LIN {X 0,Y 572.938,Z 557.197,A -85,B 0,C 180,E1 -2247.891,E2 -2247.891} C_VEL
LIN {X 0,Y 572.94,Z 558.785,A -85,B 0,C 180,E1 -2249.297,E2 -2249.297} C_VEL
LIN {X 0,Y 572.938,Z 559,A -85,B 0,C 180,E1 -2250,E2 -2250} C_VEL
LIN {X 0,Y 572.946,Z 558.187,A -85,B 0,C 180,E1 -2251.406,E2 -2251.406} C_VEL
LIN {X 0,Y 572.938,Z 557.2,A -85,B 0,C 180,E1 -2252.109,E2 -2252.109} C_VEL
LIN {X 0,Y 572.959,Z 555.811,A -85,B 0,C 180,E1 -2252.812,E2 -2252.812} C_VEL
LIN {X 0,Y 573.014,Z 552.897,A -85,B 0,C 180,E1 -2253.868,E2 -2253.868} C_VEL
LIN {X 0,Y 572.963,Z 548.95,A -85,B 0,C 180,E1 -2254.925,E2 -2254.925} C_VEL
LIN {X 0,Y 573.068,Z 542.878,A -85,B 0,C 180,E1 -2256.16,E2 -2256.16} C_VEL
LIN {X 0,Y 573.119,Z 536.24,A -85,B 0,C 180,E1 -2257.22,E2 -2257.22} C_VEL
LIN {X 0,Y 573.192,Z 527.993,A -85,B 0,C 180,E1 -2258.283,E2 -2258.283} C_VEL
LIN {X 0,Y 573.319,Z 517.605,A -85,B 0,C 180,E1 -2259.347,E2 -2259.347} C_VEL
LIN {X 0,Y 573.431,Z 507.929,A -85,B 0,C 180,E1 -2260.147,E2 -2260.147} C_VEL
LIN {X 0,Y 573.549,Z 497.407,A -85,B 0,C 180,E1 -2260.854,E2 -2260.854} C_VEL
LIN {X 0,Y 573.652,Z 486.294,A -85,B 0,C 180,E1 -2261.447,E2 -2261.447} C_VEL
LIN {X 0,Y 573.694,Z 474.482,A -85,B 0,C 180,E1 -2261.93,E2 -2261.93} C_VEL
LIN {X 0,Y 573.799,Z 461.448,A -85,B 0,C 180,E1 -2262.309,E2 -2262.309} C_VEL
LIN {X 0,Y 573.915,Z 449.111,A -85,B 0,C 180,E1 -2262.531,E2 -2262.531} C_VEL
LIN {X 0,Y 573.909,Z 350.304,A -85,B 0,C 180,E1 -2263.775,E2 -2263.775} C_VEL
LIN {X 0,Y 573.398,Z 346.616,A -85,B 0,C 180,E1 -2263.85,E2 -2263.85} C_VEL
LIN {X 0,Y 573.568,Z 326.122,A -85,B 0,C 180,E1 -2266.727,E2 -2266.727} C_VEL
LIN {X 0,Y 573.803,Z 305.614,A -85,B 0,C 180,E1 -2269.646,E2 -2269.646} C_VEL
LIN {X 0,Y 574.043,Z 285.773,A -85,B 0,C 180,E1 -2272.494,E2 -2272.494} C_VEL
LIN {X 0,Y 573.587,Z 280.817,A -85,B 0,C 180,E1 -2273.226,E2 -2273.226} C_VEL
LIN {X 0,Y 573.252,Z 279.081,A -85,B 0,C 180,E1 -2273.496,E2 -2273.496} C_VEL
LIN {X 0,Y 573.261,Z 279.078,A -85,B 0,C 180,E1 -2276.189,E2 -2276.189} C_VEL
LIN {X 0,Y 573.237,Z 279.077,A -85,B 0,C 180,E1 -2278.564,E2 -2278.564} C_VEL
LIN {X 0,Y 573.226,Z 279.075,A -85,B 0,C 180,E1 -2280.993,E2 -2280.993} C_VEL
LIN {X 0,Y 573.262,Z 279.072,A -85,B 0,C 180,E1 -2283.523,E2 -2283.523} C_VEL
LIN {X 0,Y 573.213,Z 279.084,A -85,B 0,C 180,E1 -2286.051,E2 -2286.051} C_VEL
LIN {X 0,Y 573.24,Z 279.077,A -85,B 0,C 180,E1 -2288.701,E2 -2288.701} C_VEL
LIN {X 0,Y 573.252,Z 279.072,A -85,B 0,C 180,E1 -2291.595,E2 -2291.595} C_VEL
LIN {X 0,Y 573.226,Z 279.083,A -85,B 0,C 180,E1 -2294.334,E2 -2294.334} C_VEL
LIN {X 0,Y 573.238,Z 279.074,A -85,B 0,C 180,E1 -2297.358,E2 -2297.358} C_VEL
LIN {X 0,Y 573.237,Z 279.08,A -85,B 0,C 180,E1 -2300.392,E2 -2300.392} C_VEL
LIN {X 0,Y 573.25,Z 279.076,A -85,B 0,C 180,E1 -2303.077,E2 -2303.077} C_VEL
LIN {X 0,Y 573.263,Z 279.07,A -85,B 0,C 180,E1 -2305.671,E2 -2305.671} C_VEL
LIN {X 0,Y 573.245,Z 279.074,A -85,B 0,C 180,E1 -2308.185,E2 -2308.185} C_VEL
LIN {X 0,Y 573.261,Z 279.076,A -85,B 0,C 180,E1 -2310.634,E2 -2310.634} C_VEL
LIN {X 0,Y 573.248,Z 279.083,A -85,B 0,C 180,E1 -2313.024,E2 -2313.024} C_VEL
LIN {X 0,Y 573.271,Z 279.075,A -85,B 0,C 180,E1 -2315.366,E2 -2315.366} C_VEL
LIN {X 0,Y 573.223,Z 279.076,A -85,B 0,C 180,E1 -2318.419,E2 -2318.419} C_VEL
LIN {X 0,Y 573.274,Z 279.072,A -85,B 0,C 180,E1 -2320.728,E2 -2320.728} C_VEL
LIN {X 0,Y 573.244,Z 279.077,A -85,B 0,C 180,E1 -2323.621,E2 -2323.621} C_VEL
LIN {X 0,Y 573.267,Z 279.073,A -85,B 0,C 180,E1 -2325.807,E2 -2325.807} C_VEL
LIN {X 0,Y 573.257,Z 279.072,A -85,B 0,C 180,E1 -2328.745,E2 -2328.745} C_VEL
LIN {X 0,Y 573.284,Z 279.078,A -85,B 0,C 180,E1 -2331.54,E2 -2331.54} C_VEL
LIN {X 0,Y 573.284,Z 279.068,A -85,B 0,C 180,E1 -2334.372,E2 -2334.372} C_VEL
LIN {X 0,Y 573.297,Z 279.073,A -85,B 0,C 180,E1 -2337.892,E2 -2337.892} C_VEL
LIN {X 0,Y 573.321,Z 279.063,A -85,B 0,C 180,E1 -2340.702,E2 -2340.702} C_VEL
LIN {X 0,Y 573.238,Z 279.079,A -85,B 0,C 180,E1 -2343.514,E2 -2343.514} C_VEL
LIN {X 0,Y 573.29,Z 279.073,A -85,B 0,C 180,E1 -2345.628,E2 -2345.628} C_VEL
LIN {X 0,Y 573.277,Z 279.071,A -85,B 0,C 180,E1 -2348.459,E2 -2348.459} C_VEL
LIN {X 0,Y 573.266,Z 279.071,A -85,B 0,C 180,E1 -2351.312,E2 -2351.312} C_VEL
LIN {X 0,Y 573.253,Z 279.081,A -85,B 0,C 180,E1 -2354.193,E2 -2354.193} C_VEL
LIN {X 0,Y 573.252,Z 279.072,A -85,B 0,C 180,E1 -2357.112,E2 -2357.112} C_VEL
LIN {X 0,Y 573.235,Z 279.081,A -85,B 0,C 180,E1 -2360.077,E2 -2360.077} C_VEL
LIN {X 0,Y 573.227,Z 279.086,A -85,B 0,C 180,E1 -2362.338,E2 -2362.338} C_VEL
LIN {X 0,Y 573.24,Z 279.077,A -85,B 0,C 180,E1 -2364.37,E2 -2364.37} C_VEL
LIN {X 0,Y 572.61,Z 279.158,A -85,B 0,C 180,E1 -2364.956,E2 -2364.956} C_VEL
LIN {X 0,Y 569.752,Z 279.513,A -85,B 0,C 180,E1 -2365.907,E2 -2365.907} C_VEL
LIN {X 0,Y 567.309,Z 279.819,A -85,B 0,C 180,E1 -2366.672,E2 -2366.672} C_VEL
LIN {X 0,Y 566.252,Z 279.944,A -85,B 0,C 180,E1 -2367.264,E2 -2367.264} C_VEL
LIN {X 0,Y 566.163,Z 279.955,A -85,B 0,C 180,E1 -2367.464,E2 -2367.464} C_VEL
LIN {X 0,Y 566.194,Z 279.951,A -85,B 0,C 180,E1 -2369.769,E2 -2369.769} C_VEL
LIN {X 0,Y 566.198,Z 279.958,A -85,B 0,C 180,E1 -2372.43,E2 -2372.43} C_VEL
LIN {X 0,Y 566.173,Z 279.959,A -85,B 0,C 180,E1 -2374.99,E2 -2374.99} C_VEL
LIN {X 0,Y 566.19,Z 279.952,A -85,B 0,C 180,E1 -2377.461,E2 -2377.461} C_VEL
LIN {X 0,Y 566.201,Z 279.952,A -85,B 0,C 180,E1 -2380.2,E2 -2380.2} C_VEL
LIN {X 0,Y 566.192,Z 279.959,A -85,B 0,C 180,E1 -2383.055,E2 -2383.055} C_VEL
LIN {X 0,Y 566.188,Z 279.951,A -85,B 0,C 180,E1 -2386.05,E2 -2386.05} C_VEL
LIN {X 0,Y 566.198,Z 279.959,A -85,B 0,C 180,E1 -2389.215,E2 -2389.215} C_VEL
LIN {X 0,Y 566.175,Z 279.956,A -85,B 0,C 180,E1 -2391.637,E2 -2391.637} C_VEL
LIN {X 0,Y 566.157,Z 279.955,A -85,B 0,C 180,E1 -2394.308,E2 -2394.308} C_VEL
LIN {X 0,Y 566.194,Z 279.955,A -85,B 0,C 180,E1 -2396.897,E2 -2396.897} C_VEL
LIN {X 0,Y 566.159,Z 279.965,A -85,B 0,C 180,E1 -2399.407,E2 -2399.407} C_VEL
LIN {X 0,Y 566.184,Z 279.955,A -85,B 0,C 180,E1 -2401.856,E2 -2401.856} C_VEL
LIN {X 0,Y 566.18,Z 279.953,A -85,B 0,C 180,E1 -2404.25,E2 -2404.25} C_VEL
LIN {X 0,Y 566.172,Z 279.961,A -85,B 0,C 180,E1 -2407.369,E2 -2407.369} C_VEL
LIN {X 0,Y 566.202,Z 279.96,A -85,B 0,C 180,E1 -2409.663,E2 -2409.663} C_VEL
LIN {X 0,Y 566.175,Z 279.96,A -85,B 0,C 180,E1 -2411.921,E2 -2411.921} C_VEL
LIN {X 0,Y 566.188,Z 279.952,A -85,B 0,C 180,E1 -2414.891,E2 -2414.891} C_VEL
LIN {X 0,Y 566.209,Z 279.96,A -85,B 0,C 180,E1 -2417.819,E2 -2417.819} C_VEL
LIN {X 0,Y 566.179,Z 279.957,A -85,B 0,C 180,E1 -2420.714,E2 -2420.714} C_VEL
LIN {X 0,Y 566.192,Z 280.141,A -85,B 0,C 180,E1 -2420.894,E2 -2420.894} C_VEL
LIN {X 0,Y 566.476,Z 285.072,A -85,B 0,C 180,E1 -2421.798,E2 -2421.798} C_VEL
LIN {X 0,Y 566.29,Z 300.723,A -85,B 0,C 180,E1 -2424.66,E2 -2424.66} C_VEL
LIN {X 0,Y 566.196,Z 308.354,A -85,B 0,C 180,E1 -2426.041,E2 -2426.041} C_VEL
LIN {X 0,Y 567.175,Z 314.722,A -85,B 0,C 180,E1 -2426.159,E2 -2426.159} C_VEL
LIN {X 0,Y 566.923,Z 414.925,A -85,B 0,C 180,E1 -2427.447,E2 -2427.447} C_VEL
LIN {X 0,Y 566.838,Z 428.007,A -85,B 0,C 180,E1 -2427.758,E2 -2427.758} C_VEL
LIN {X 0,Y 566.75,Z 441.122,A -85,B 0,C 180,E1 -2428.224,E2 -2428.224} C_VEL
LIN {X 0,Y 566.61,Z 452.221,A -85,B 0,C 180,E1 -2428.756,E2 -2428.756} C_VEL
LIN {X 0,Y 566.39,Z 463.741,A -85,B 0,C 180,E1 -2429.467,E2 -2429.467} C_VEL
LIN {X 0,Y 566.297,Z 474.096,A -85,B 0,C 180,E1 -2430.267,E2 -2430.267} C_VEL
LIN {X 0,Y 566.199,Z 482.596,A -85,B 0,C 180,E1 -2431.067,E2 -2431.067} C_VEL
LIN {X 0,Y 566.087,Z 490.471,A -85,B 0,C 180,E1 -2431.957,E2 -2431.957} C_VEL
LIN {X 0,Y 566.044,Z 498.203,A -85,B 0,C 180,E1 -2433.025,E2 -2433.025} C_VEL
LIN {X 0,Y 565.964,Z 505.322,A -85,B 0,C 180,E1 -2434.273,E2 -2434.273} C_VEL
LIN {X 0,Y 565.923,Z 510.091,A -85,B 0,C 180,E1 -2435.344,E2 -2435.344} C_VEL
LIN {X 0,Y 565.944,Z 514.182,A -85,B 0,C 180,E1 -2436.56,E2 -2436.56} C_VEL
LIN {X 0,Y 565.876,Z 517.108,A -85,B 0,C 180,E1 -2437.852,E2 -2437.852} C_VEL
LIN {X 0,Y 565.851,Z 518.129,A -85,B 0,C 180,E1 -2438.572,E2 -2438.572} C_VEL
LIN {X 0,Y 565.88,Z 518.998,A -85,B 0,C 180,E1 -2440.013,E2 -2440.013} C_VEL
LIN {X 0,Y 565.9,Z 518.518,A -85,B 0,C 180,E1 -2441.154,E2 -2441.154} C_VEL
LIN {X 0,Y 565.867,Z 517.182,A -85,B 0,C 180,E1 -2442.189,E2 -2442.189} C_VEL
LIN {X 0,Y 565.852,Z 515.747,A -85,B 0,C 180,E1 -2442.919,E2 -2442.919} C_VEL
LIN {X 0,Y 565.916,Z 512.727,A -85,B 0,C 180,E1 -2444.015,E2 -2444.015} C_VEL
LIN {X 0,Y 565.947,Z 508.595,A -85,B 0,C 180,E1 -2445.117,E2 -2445.117} C_VEL
LIN {X 0,Y 565.955,Z 502.16,A -85,B 0,C 180,E1 -2446.41,E2 -2446.41} C_VEL
LIN {X 0,Y 566.076,Z 495.095,A -85,B 0,C 180,E1 -2447.522,E2 -2447.522} C_VEL
LIN {X 0,Y 566.142,Z 487.805,A -85,B 0,C 180,E1 -2448.455,E2 -2448.455} C_VEL
LIN {X 0,Y 566.249,Z 477.889,A -85,B 0,C 180,E1 -2449.484,E2 -2449.484} C_VEL
LIN {X 0,Y 566.378,Z 467.78,A -85,B 0,C 180,E1 -2450.331,E2 -2450.331} C_VEL
LIN {X 0,Y 566.526,Z 456.576,A -85,B 0,C 180,E1 -2451.085,E2 -2451.085} C_VEL
LIN {X 0,Y 566.679,Z 444.223,A -85,B 0,C 180,E1 -2451.73,E2 -2451.73} C_VEL
LIN {X 0,Y 566.776,Z 431.645,A -85,B 0,C 180,E1 -2452.222,E2 -2452.222} C_VEL
LIN {X 0,Y 566.799,Z 419.367,A -85,B 0,C 180,E1 -2452.557,E2 -2452.557} C_VEL
LIN {X 0,Y 566.916,Z 402.556,A -85,B 0,C 180,E1 -2452.817,E2 -2452.817} C_VEL
LIN {X 0,Y 567.066,Z 313.669,A -85,B 0,C 180,E1 -2453.947,E2 -2453.947} C_VEL
LIN {X 0,Y 566.196,Z 308.415,A -85,B 0,C 180,E1 -2454.038,E2 -2454.038} C_VEL
LIN {X 0,Y 566.375,Z 293.793,A -85,B 0,C 180,E1 -2456.693,E2 -2456.693} C_VEL
LIN {X 0,Y 566.454,Z 281.463,A -85,B 0,C 180,E1 -2458.939,E2 -2458.939} C_VEL
LIN {X 0,Y 566.256,Z 279.95,A -85,B 0,C 180,E1 -2459.255,E2 -2459.255} C_VEL
LIN {X 0,Y 566.204,Z 279.959,A -85,B 0,C 180,E1 -2462.43,E2 -2462.43} C_VEL
LIN {X 0,Y 566.178,Z 279.955,A -85,B 0,C 180,E1 -2464.989,E2 -2464.989} C_VEL
LIN {X 0,Y 566.195,Z 279.95,A -85,B 0,C 180,E1 -2467.461,E2 -2467.461} C_VEL
LIN {X 0,Y 566.206,Z 279.956,A -85,B 0,C 180,E1 -2470.199,E2 -2470.199} C_VEL
LIN {X 0,Y 566.199,Z 279.954,A -85,B 0,C 180,E1 -2473.054,E2 -2473.054} C_VEL
LIN {X 0,Y 566.193,Z 279.953,A -85,B 0,C 180,E1 -2476.049,E2 -2476.049} C_VEL
LIN {X 0,Y 566.203,Z 279.953,A -85,B 0,C 180,E1 -2479.215,E2 -2479.215} C_VEL
LIN {X 0,Y 566.185,Z 279.952,A -85,B 0,C 180,E1 -2481.637,E2 -2481.637} C_VEL
LIN {X 0,Y 566.161,Z 279.956,A -85,B 0,C 180,E1 -2484.308,E2 -2484.308} C_VEL
LIN {X 0,Y 566.218,Z 279.956,A -85,B 0,C 180,E1 -2486.898,E2 -2486.898} C_VEL
LIN {X 0,Y 566.18,Z 279.957,A -85,B 0,C 180,E1 -2489.407,E2 -2489.407} C_VEL
LIN {X 0,Y 566.21,Z 279.948,A -85,B 0,C 180,E1 -2491.857,E2 -2491.857} C_VEL
LIN {X 0,Y 566.212,Z 279.948,A -85,B 0,C 180,E1 -2494.251,E2 -2494.251} C_VEL
LIN {X 0,Y 566.172,Z 279.954,A -85,B 0,C 180,E1 -2496.718,E2 -2496.718} C_VEL
LIN {X 0,Y 566.207,Z 279.954,A -85,B 0,C 180,E1 -2499.663,E2 -2499.663} C_VEL
LIN {X 0,Y 566.198,Z 279.951,A -85,B 0,C 180,E1 -2502.668,E2 -2502.668} C_VEL
LIN {X 0,Y 566.233,Z 279.957,A -85,B 0,C 180,E1 -2505.627,E2 -2505.627} C_VEL
LIN {X 0,Y 566.233,Z 279.945,A -85,B 0,C 180,E1 -2508.675,E2 -2508.675} C_VEL
LIN {X 0,Y 566.226,Z 279.952,A -85,B 0,C 180,E1 -2511.434,E2 -2511.434} C_VEL
LIN {X 0,Y 566.256,Z 279.946,A -85,B 0,C 180,E1 -2514.302,E2 -2514.302} C_VEL
LIN {X 0,Y 566.281,Z 279.949,A -85,B 0,C 180,E1 -2517.866,E2 -2517.866} C_VEL
LIN {X 0,Y 566.299,Z 279.939,A -85,B 0,C 180,E1 -2520.711,E2 -2520.711} C_VEL
LIN {X 0,Y 566.27,Z 279.941,A -85,B 0,C 180,E1 -2522.846,E2 -2522.846} C_VEL
LIN {X 0,Y 566.256,Z 279.946,A -85,B 0,C 180,E1 -2525.698,E2 -2525.698} C_VEL
LIN {X 0,Y 566.226,Z 279.953,A -85,B 0,C 180,E1 -2528.566,E2 -2528.566} C_VEL
LIN {X 0,Y 566.242,Z 279.944,A -85,B 0,C 180,E1 -2531.454,E2 -2531.454} C_VEL
LIN {X 0,Y 566.234,Z 279.956,A -85,B 0,C 180,E1 -2534.507,E2 -2534.507} C_VEL
LIN {X 0,Y 566.199,Z 279.951,A -85,B 0,C 180,E1 -2537.332,E2 -2537.332} C_VEL
LIN {X 0,Y 566.207,Z 279.954,A -85,B 0,C 180,E1 -2540.338,E2 -2540.338} C_VEL
LIN {X 0,Y 566.173,Z 279.956,A -85,B 0,C 180,E1 -2543.282,E2 -2543.282} C_VEL
LIN {X 0,Y 566.214,Z 279.948,A -85,B 0,C 180,E1 -2545.749,E2 -2545.749} C_VEL
LIN {X 0,Y 566.203,Z 279.95,A -85,B 0,C 180,E1 -2548.202,E2 -2548.202} C_VEL
LIN {X 0,Y 566.191,Z 279.96,A -85,B 0,C 180,E1 -2551.077,E2 -2551.077} C_VEL
LIN {X 0,Y 566.212,Z 279.95,A -85,B 0,C 180,E1 -2553.734,E2 -2553.734} C_VEL
LIN {X 0,Y 566.2,Z 279.951,A -85,B 0,C 180,E1 -2556.57,E2 -2556.57} C_VEL
LIN {X 0,Y 566.216,Z 279.949,A -85,B 0,C 180,E1 -2559.686,E2 -2559.686} C_VEL
LIN {X 0,Y 566.203,Z 279.953,A -85,B 0,C 180,E1 -2562.917,E2 -2562.917} C_VEL
LIN {X 0,Y 566.195,Z 279.953,A -85,B 0,C 180,E1 -2566.049,E2 -2566.049} C_VEL
LIN {X 0,Y 566.205,Z 279.955,A -85,B 0,C 180,E1 -2569.215,E2 -2569.215} C_VEL
LIN {X 0,Y 566.187,Z 279.962,A -85,B 0,C 180,E1 -2571.637,E2 -2571.637} C_VEL
LIN {X 0,Y 566.163,Z 279.957,A -85,B 0,C 180,E1 -2574.308,E2 -2574.308} C_VEL
LIN {X 0,Y 566.207,Z 279.95,A -85,B 0,C 180,E1 -2576.897,E2 -2576.897} C_VEL
LIN {X 0,Y 566.183,Z 279.957,A -85,B 0,C 180,E1 -2579.407,E2 -2579.407} C_VEL
LIN {X 0,Y 566.197,Z 279.961,A -85,B 0,C 180,E1 -2581.857,E2 -2581.857} C_VEL
LIN {X 0,Y 566.211,Z 279.957,A -85,B 0,C 180,E1 -2584.251,E2 -2584.251} C_VEL
LIN {X 0,Y 566.227,Z 280.119,A -85,B 0,C 180,E1 -2586.404,E2 -2586.404} C_VEL
LIN {X 0,Y 567.053,Z 285.451,A -85,B 0,C 180,E1 -2587.213,E2 -2587.213} C_VEL
LIN {X 0,Y 566.869,Z 303.945,A -85,B 0,C 180,E1 -2589.877,E2 -2589.877} C_VEL
LIN {X 0,Y 566.611,Z 324.891,A -85,B 0,C 180,E1 -2592.885,E2 -2592.885} C_VEL
LIN {X 0,Y 566.39,Z 346.612,A -85,B 0,C 180,E1 -2595.974,E2 -2595.974} C_VEL
LIN {X 0,Y 567.217,Z 352.273,A -85,B 0,C 180,E1 -2596.084,E2 -2596.084} C_VEL
LIN {X 0,Y 566.954,Z 454.939,A -85,B 0,C 180,E1 -2597.403,E2 -2597.403} C_VEL
LIN {X 0,Y 566.847,Z 467.451,A -85,B 0,C 180,E1 -2597.696,E2 -2597.696} C_VEL
LIN {X 0,Y 566.724,Z 480.373,A -85,B 0,C 180,E1 -2598.148,E2 -2598.148} C_VEL
LIN {X 0,Y 566.631,Z 492.046,A -85,B 0,C 180,E1 -2598.702,E2 -2598.702} C_VEL
LIN {X 0,Y 566.488,Z 502.905,A -85,B 0,C 180,E1 -2599.365,E2 -2599.365} C_VEL
LIN {X 0,Y 566.33,Z 513.537,A -85,B 0,C 180,E1 -2600.175,E2 -2600.175} C_VEL
LIN {X 0,Y 566.206,Z 523.081,A -85,B 0,C 180,E1 -2601.074,E2 -2601.074} C_VEL
LIN {X 0,Y 566.111,Z 530.959,A -85,B 0,C 180,E1 -2601.971,E2 -2601.971} C_VEL
LIN {X 0,Y 566.004,Z 538.621,A -85,B 0,C 180,E1 -2603.046,E2 -2603.046} C_VEL
LIN {X 0,Y 566.004,Z 545.679,A -85,B 0,C 180,E1 -2604.299,E2 -2604.299} C_VEL
LIN {X 0,Y 565.933,Z 550.371,A -85,B 0,C 180,E1 -2605.37,E2 -2605.37} C_VEL
LIN {X 0,Y 565.927,Z 553.957,A -85,B 0,C 180,E1 -2606.44,E2 -2606.44} C_VEL
LIN {X 0,Y 565.878,Z 555.807,A -85,B 0,C 180,E1 -2607.152,E2 -2607.152} C_VEL
LIN {X 0,Y 565.845,Z 558.185,A -85,B 0,C 180,E1 -2608.576,E2 -2608.576} C_VEL
LIN {X 0,Y 565.839,Z 559,A -85,B 0,C 180,E1 -2610,E2 -2610} C_VEL
LIN {X 0,Y 565.845,Z 558.186,A -85,B 0,C 180,E1 -2611.423,E2 -2611.423} C_VEL
LIN {X 0,Y 565.878,Z 555.811,A -85,B 0,C 180,E1 -2612.847,E2 -2612.847} C_VEL
LIN {X 0,Y 565.926,Z 552.896,A -85,B 0,C 180,E1 -2613.916,E2 -2613.916} C_VEL
LIN {X 0,Y 565.878,Z 548.95,A -85,B 0,C 180,E1 -2614.987,E2 -2614.987} C_VEL
LIN {X 0,Y 566.004,Z 543.869,A -85,B 0,C 180,E1 -2616.058,E2 -2616.058} C_VEL
LIN {X 0,Y 566.04,Z 537.47,A -85,B 0,C 180,E1 -2617.132,E2 -2617.132} C_VEL
LIN {X 0,Y 566.128,Z 529.481,A -85,B 0,C 180,E1 -2618.207,E2 -2618.207} C_VEL
LIN {X 0,Y 566.228,Z 521.338,A -85,B 0,C 180,E1 -2619.105,E2 -2619.105} C_VEL
LIN {X 0,Y 566.336,Z 511.404,A -85,B 0,C 180,E1 -2620.005,E2 -2620.005} C_VEL
LIN {X 0,Y 566.543,Z 500.307,A -85,B 0,C 180,E1 -2620.806,E2 -2620.806} C_VEL
LIN {X 0,Y 566.64,Z 489.182,A -85,B 0,C 180,E1 -2621.446,E2 -2621.446} C_VEL
LIN {X 0,Y 566.757,Z 476.99,A -85,B 0,C 180,E1 -2621.987,E2 -2621.987} C_VEL
LIN {X 0,Y 566.868,Z 464.19,A -85,B 0,C 180,E1 -2622.394,E2 -2622.394} C_VEL
LIN {X 0,Y 566.986,Z 450.626,A -85,B 0,C 180,E1 -2622.664,E2 -2622.664} C_VEL
LIN {X 0,Y 567.103,Z 351.644,A -85,B 0,C 180,E1 -2623.927,E2 -2623.927} C_VEL
LIN {X 0,Y 566.406,Z 346.616,A -85,B 0,C 180,E1 -2624.025,E2 -2624.025} C_VEL
LIN {X 0,Y 566.606,Z 324.043,A -85,B 0,C 180,E1 -2627.237,E2 -2627.237} C_VEL
LIN {X 0,Y 566.868,Z 303.962,A -85,B 0,C 180,E1 -2630.123,E2 -2630.123} C_VEL
LIN {X 0,Y 567.088,Z 285.517,A -85,B 0,C 180,E1 -2632.785,E2 -2632.785} C_VEL
LIN {X 0,Y 566.214,Z 279.959,A -85,B 0,C 180,E1 -2633.645,E2 -2633.645} C_VEL
LIN {X 0,Y 566.21,Z 279.958,A -85,B 0,C 180,E1 -2635.749,E2 -2635.749} C_VEL
LIN {X 0,Y 566.203,Z 279.959,A -85,B 0,C 180,E1 -2638.201,E2 -2638.201} C_VEL
LIN {X 0,Y 566.191,Z 279.951,A -85,B 0,C 180,E1 -2641.076,E2 -2641.076} C_VEL
LIN {X 0,Y 566.211,Z 279.952,A -85,B 0,C 180,E1 -2643.734,E2 -2643.734} C_VEL
LIN {X 0,Y 566.199,Z 279.956,A -85,B 0,C 180,E1 -2646.569,E2 -2646.569} C_VEL
LIN {X 0,Y 566.213,Z 279.95,A -85,B 0,C 180,E1 -2649.685,E2 -2649.685} C_VEL
LIN {X 0,Y 566.212,Z 279.954,A -85,B 0,C 180,E1 -2652.087,E2 -2652.087} C_VEL
LIN {X 0,Y 566.169,Z 279.956,A -85,B 0,C 180,E1 -2655.035,E2 -2655.035} C_VEL
LIN {X 0,Y 566.216,Z 279.951,A -85,B 0,C 180,E1 -2658.135,E2 -2658.135} C_VEL
LIN {X 0,Y 566.212,Z 279.958,A -85,B 0,C 180,E1 -2660.726,E2 -2660.726} C_VEL
LIN {X 0,Y 566.182,Z 279.952,A -85,B 0,C 180,E1 -2663.787,E2 -2663.787} C_VEL
LIN {X 0,Y 566.208,Z 279.951,A -85,B 0,C 180,E1 -2666.265,E2 -2666.265} C_VEL
LIN {X 0,Y 566.196,Z 279.961,A -85,B 0,C 180,E1 -2668.922,E2 -2668.922} C_VEL
LIN {X 0,Y 566.207,Z 279.949,A -85,B 0,C 180,E1 -2671.857,E2 -2671.857} C_VEL
LIN {X 0,Y 566.211,Z 279.949,A -85,B 0,C 180,E1 -2674.251,E2 -2674.251} C_VEL
LIN {X 0,Y 566.187,Z 279.956,A -85,B 0,C 180,E1 -2676.713,E2 -2676.713} C_VEL
LIN {X 0,Y 566.208,Z 279.952,A -85,B 0,C 180,E1 -2679.662,E2 -2679.662} C_VEL
LIN {X 0,Y 566.194,Z 279.953,A -85,B 0,C 180,E1 -2682.668,E2 -2682.668} C_VEL
LIN {X 0,Y 566.228,Z 279.952,A -85,B 0,C 180,E1 -2685.626,E2 -2685.626} C_VEL
LIN {X 0,Y 566.229,Z 279.947,A -85,B 0,C 180,E1 -2688.675,E2 -2688.675} C_VEL
LIN {X 0,Y 566.228,Z 279.957,A -85,B 0,C 180,E1 -2691.434,E2 -2691.434} C_VEL
LIN {X 0,Y 566.251,Z 279.944,A -85,B 0,C 180,E1 -2694.301,E2 -2694.301} C_VEL
LIN {X 0,Y 566.269,Z 279.949,A -85,B 0,C 180,E1 -2697.866,E2 -2697.866} C_VEL
LIN {X 0,Y 566.292,Z 279.939,A -85,B 0,C 180,E1 -2700.711,E2 -2700.711} C_VEL
LIN {X 0,Y 566.263,Z 279.942,A -85,B 0,C 180,E1 -2702.845,E2 -2702.845} C_VEL
LIN {X 0,Y 566.256,Z 279.951,A -85,B 0,C 180,E1 -2705.698,E2 -2705.698} C_VEL
LIN {X 0,Y 566.221,Z 279.949,A -85,B 0,C 180,E1 -2708.566,E2 -2708.566} C_VEL
LIN {X 0,Y 566.236,Z 279.947,A -85,B 0,C 180,E1 -2711.454,E2 -2711.454} C_VEL
LIN {X 0,Y 566.217,Z 279.952,A -85,B 0,C 180,E1 -2714.502,E2 -2714.502} C_VEL
LIN {X 0,Y 566.192,Z 279.951,A -85,B 0,C 180,E1 -2717.332,E2 -2717.332} C_VEL
LIN {X 0,Y 566.201,Z 279.96,A -85,B 0,C 180,E1 -2720.337,E2 -2720.337} C_VEL
LIN {X 0,Y 566.163,Z 279.955,A -85,B 0,C 180,E1 -2723.281,E2 -2723.281} C_VEL
LIN {X 0,Y 566.206,Z 279.95,A -85,B 0,C 180,E1 -2725.749,E2 -2725.749} C_VEL
LIN {X 0,Y 566.163,Z 279.955,A -85,B 0,C 180,E1 -2727.464,E2 -2727.464} C_VEL
LIN {X 0,Y 565.491,Z 280.044,A -85,B 0,C 180,E1 -2728.058,E2 -2728.058} C_VEL
LIN {X 0,Y 562.639,Z 280.396,A -85,B 0,C 180,E1 -2729.022,E2 -2729.022} C_VEL
LIN {X 0,Y 560.238,Z 280.696,A -85,B 0,C 180,E1 -2729.798,E2 -2729.798} C_VEL
LIN {X 0,Y 559.213,Z 280.828,A -85,B 0,C 180,E1 -2730.397,E2 -2730.397} C_VEL
LIN {X 0,Y 559.132,Z 280.833,A -85,B 0,C 180,E1 -2730.6,E2 -2730.6} C_VEL
LIN {X 0,Y 559.147,Z 280.838,A -85,B 0,C 180,E1 -2732.716,E2 -2732.716} C_VEL
LIN {X 0,Y 559.121,Z 280.833,A -85,B 0,C 180,E1 -2735.324,E2 -2735.324} C_VEL
LIN {X 0,Y 559.126,Z 280.832,A -85,B 0,C 180,E1 -2738.018,E2 -2738.018} C_VEL
LIN {X 0,Y 559.149,Z 280.839,A -85,B 0,C 180,E1 -2740.813,E2 -2740.813} C_VEL
LIN {X 0,Y 559.132,Z 280.831,A -85,B 0,C 180,E1 -2743.735,E2 -2743.735} C_VEL
LIN {X 0,Y 559.135,Z 280.837,A -85,B 0,C 180,E1 -2746.805,E2 -2746.805} C_VEL
LIN {X 0,Y 559.149,Z 280.837,A -85,B 0,C 180,E1 -2749.188,E2 -2749.188} C_VEL
LIN {X 0,Y 559.125,Z 280.832,A -85,B 0,C 180,E1 -2751.982,E2 -2751.982} C_VEL
LIN {X 0,Y 559.127,Z 280.835,A -85,B 0,C 180,E1 -2754.788,E2 -2754.788} C_VEL
LIN {X 0,Y 559.148,Z 280.838,A -85,B 0,C 180,E1 -2757.366,E2 -2757.366} C_VEL
LIN {X 0,Y 559.108,Z 280.834,A -85,B 0,C 180,E1 -2760.15,E2 -2760.15} C_VEL
LIN {X 0,Y 559.121,Z 280.832,A -85,B 0,C 180,E1 -2762.285,E2 -2762.285} C_VEL
LIN {X 0,Y 559.135,Z 280.831,A -85,B 0,C 180,E1 -2764.823,E2 -2764.823} C_VEL
LIN {X 0,Y 559.135,Z 280.836,A -85,B 0,C 180,E1 -2767.847,E2 -2767.847} C_VEL
LIN {X 0,Y 559.191,Z 280.823,A -85,B 0,C 180,E1 -2770.495,E2 -2770.495} C_VEL
LIN {X 0,Y 559.143,Z 280.832,A -85,B 0,C 180,E1 -2773.197,E2 -2773.197} C_VEL
LIN {X 0,Y 559.154,Z 280.833,A -85,B 0,C 180,E1 -2776.184,E2 -2776.184} C_VEL
LIN {X 0,Y 559.163,Z 280.829,A -85,B 0,C 180,E1 -2779.133,E2 -2779.133} C_VEL
LIN {X 0,Y 559.136,Z 280.872,A -85,B 0,C 180,E1 -2780.824,E2 -2780.824} C_VEL
LIN {X 0,Y 559.451,Z 286.635,A -85,B 0,C 180,E1 -2781.876,E2 -2781.876} C_VEL
LIN {X 0,Y 559.274,Z 301.432,A -85,B 0,C 180,E1 -2784.592,E2 -2784.592} C_VEL
LIN {X 0,Y 559.202,Z 308.679,A -85,B 0,C 180,E1 -2785.879,E2 -2785.879} C_VEL
LIN {X 0,Y 560.311,Z 315.796,A -85,B 0,C 180,E1 -2785.999,E2 -2785.999} C_VEL
LIN {X 0,Y 560.001,Z 415.633,A -85,B 0,C 180,E1 -2787.303,E2 -2787.303} C_VEL
LIN {X 0,Y 559.887,Z 429.235,A -85,B 0,C 180,E1 -2787.64,E2 -2787.64} C_VEL
LIN {X 0,Y 559.787,Z 441.991,A -85,B 0,C 180,E1 -2788.112,E2 -2788.112} C_VEL
LIN {X 0,Y 559.557,Z 454.44,A -85,B 0,C 180,E1 -2788.741,E2 -2788.741} C_VEL
LIN {X 0,Y 559.363,Z 465.539,A -85,B 0,C 180,E1 -2789.46,E2 -2789.46} C_VEL
LIN {X 0,Y 559.267,Z 474.533,A -85,B 0,C 180,E1 -2790.18,E2 -2790.18} C_VEL
LIN {X 0,Y 559.136,Z 483.802,A -85,B 0,C 180,E1 -2791.081,E2 -2791.081} C_VEL
LIN {X 0,Y 558.995,Z 492.827,A -85,B 0,C 180,E1 -2792.162,E2 -2792.162} C_VEL
LIN {X 0,Y 558.898,Z 500.108,A -85,B 0,C 180,E1 -2793.244,E2 -2793.244} C_VEL
LIN {X 0,Y 558.892,Z 505.958,A -85,B 0,C 180,E1 -2794.327,E2 -2794.327} C_VEL
LIN {X 0,Y 558.848,Z 510.592,A -85,B 0,C 180,E1 -2795.412,E2 -2795.412} C_VEL
LIN {X 0,Y 558.843,Z 514.241,A -85,B 0,C 180,E1 -2796.536,E2 -2796.536} C_VEL
LIN {X 0,Y 558.793,Z 515.946,A -85,B 0,C 180,E1 -2797.225,E2 -2797.225} C_VEL
LIN {X 0,Y 558.794,Z 517.306,A -85,B 0,C 180,E1 -2797.952,E2 -2797.952} C_VEL
LIN {X 0,Y 558.765,Z 518.271,A -85,B 0,C 180,E1 -2798.681,E2 -2798.681} C_VEL
LIN {X 0,Y 558.74,Z 518.842,A -85,B 0,C 180,E1 -2799.411,E2 -2799.411} C_VEL
LIN {X 0,Y 558.776,Z 518.985,A -85,B 0,C 180,E1 -2800.142,E2 -2800.142} C_VEL
LIN {X 0,Y 558.797,Z 518.504,A -85,B 0,C 180,E1 -2801.185,E2 -2801.185} C_VEL
LIN {X 0,Y 558.774,Z 516.974,A -85,B 0,C 180,E1 -2802.346,E2 -2802.346} C_VEL
LIN {X 0,Y 558.755,Z 515.428,A -85,B 0,C 180,E1 -2803.086,E2 -2803.086} C_VEL
LIN {X 0,Y 558.825,Z 511.423,A -85,B 0,C 180,E1 -2804.447,E2 -2804.447} C_VEL
LIN {X 0,Y 558.864,Z 506.335,A -85,B 0,C 180,E1 -2805.687,E2 -2805.687} C_VEL
LIN {X 0,Y 558.954,Z 500.326,A -85,B 0,C 180,E1 -2806.81,E2 -2806.81} C_VEL
LIN {X 0,Y 559.037,Z 492.742,A -85,B 0,C 180,E1 -2807.939,E2 -2807.939} C_VEL
LIN {X 0,Y 559.146,Z 484.946,A -85,B 0,C 180,E1 -2808.884,E2 -2808.884} C_VEL
LIN {X 0,Y 559.274,Z 475.408,A -85,B 0,C 180,E1 -2809.834,E2 -2809.834} C_VEL
LIN {X 0,Y 559.422,Z 464.653,A -85,B 0,C 180,E1 -2810.691,E2 -2810.691} C_VEL
LIN {X 0,Y 559.598,Z 452.715,A -85,B 0,C 180,E1 -2811.448,E2 -2811.448} C_VEL
LIN {X 0,Y 559.742,Z 442.039,A -85,B 0,C 180,E1 -2811.977,E2 -2811.977} C_VEL
LIN {X 0,Y 559.846,Z 429.64,A -85,B 0,C 180,E1 -2812.439,E2 -2812.439} C_VEL
LIN {X 0,Y 559.928,Z 416.24,A -85,B 0,C 180,E1 -2812.777,E2 -2812.777} C_VEL
LIN {X 0,Y 560.069,Z 380.623,A -85,B 0,C 180,E1 -2813.259,E2 -2813.259} C_VEL
LIN {X 0,Y 560.256,Z 314.909,A -85,B 0,C 180,E1 -2814.103,E2 -2814.103} C_VEL
LIN {X 0,Y 559.188,Z 308.333,A -85,B 0,C 180,E1 -2814.232,E2 -2814.232} C_VEL
LIN {X 0,Y 559.364,Z 293.827,A -85,B 0,C 180,E1 -2816.892,E2 -2816.892} C_VEL
LIN {X 0,Y 559.419,Z 282.433,A -85,B 0,C 180,E1 -2818.926,E2 -2818.926} C_VEL
LIN {X 0,Y 559.235,Z 280.825,A -85,B 0,C 180,E1 -2819.245,E2 -2819.245} C_VEL
LIN {X 0,Y 559.165,Z 280.833,A -85,B 0,C 180,E1 -2821.863,E2 -2821.863} C_VEL
LIN {X 0,Y 559.142,Z 280.839,A -85,B 0,C 180,E1 -2824.445,E2 -2824.445} C_VEL
LIN {X 0,Y 559.14,Z 280.829,A -85,B 0,C 180,E1 -2827.108,E2 -2827.108} C_VEL
LIN {X 0,Y 559.159,Z 280.83,A -85,B 0,C 180,E1 -2829.942,E2 -2829.942} C_VEL
LIN {X 0,Y 559.156,Z 280.836,A -85,B 0,C 180,E1 -2832.744,E2 -2832.744} C_VEL
LIN {X 0,Y 559.146,Z 280.829,A -85,B 0,C 180,E1 -2835.761,E2 -2835.761} C_VEL
LIN {X 0,Y 559.162,Z 280.83,A -85,B 0,C 180,E1 -2838.23,E2 -2838.23} C_VEL
LIN {X 0,Y 559.174,Z 280.829,A -85,B 0,C 180,E1 -2841.192,E2 -2841.192} C_VEL
LIN {X 0,Y 559.138,Z 280.829,A -85,B 0,C 180,E1 -2843.789,E2 -2843.789} C_VEL
LIN {X 0,Y 559.161,Z 280.828,A -85,B 0,C 180,E1 -2846.425,E2 -2846.425} C_VEL
LIN {X 0,Y 559.154,Z 280.836,A -85,B 0,C 180,E1 -2848.981,E2 -2848.981} C_VEL
LIN {X 0,Y 559.167,Z 280.828,A -85,B 0,C 180,E1 -2851.619,E2 -2851.619} C_VEL
LIN {X 0,Y 559.179,Z 280.825,A -85,B 0,C 180,E1 -2853.903,E2 -2853.903} C_VEL
LIN {X 0,Y 559.141,Z 280.828,A -85,B 0,C 180,E1 -2856.571,E2 -2856.571} C_VEL
LIN {X 0,Y 559.176,Z 280.835,A -85,B 0,C 180,E1 -2859.395,E2 -2859.395} C_VEL
LIN {X 0,Y 559.142,Z 280.836,A -85,B 0,C 180,E1 -2861.686,E2 -2861.686} C_VEL
LIN {X 0,Y 559.165,Z 280.829,A -85,B 0,C 180,E1 -2863.948,E2 -2863.948} C_VEL
LIN {X 0,Y 559.17,Z 280.828,A -85,B 0,C 180,E1 -2866.184,E2 -2866.184} C_VEL
LIN {X 0,Y 559.192,Z 280.824,A -85,B 0,C 180,E1 -2869.134,E2 -2869.134} C_VEL
LIN {X 0,Y 559.203,Z 280.827,A -85,B 0,C 180,E1 -2872.054,E2 -2872.054} C_VEL
LIN {X 0,Y 559.249,Z 280.816,A -85,B 0,C 180,E1 -2874.953,E2 -2874.953} C_VEL
LIN {X 0,Y 559.252,Z 280.824,A -85,B 0,C 180,E1 -2877.84,E2 -2877.84} C_VEL
LIN {X 0,Y 559.27,Z 280.814,A -85,B 0,C 180,E1 -2880.72,E2 -2880.72} C_VEL
LIN {X 0,Y 559.236,Z 280.817,A -85,B 0,C 180,E1 -2882.882,E2 -2882.882} C_VEL
LIN {X 0,Y 559.225,Z 280.822,A -85,B 0,C 180,E1 -2885.77,E2 -2885.77} C_VEL
LIN {X 0,Y 559.185,Z 280.828,A -85,B 0,C 180,E1 -2888.675,E2 -2888.675} C_VEL
LIN {X 0,Y 559.205,Z 280.82,A -85,B 0,C 180,E1 -2891.601,E2 -2891.601} C_VEL
LIN {X 0,Y 559.2,Z 280.83,A -85,B 0,C 180,E1 -2894.596,E2 -2894.596} C_VEL
LIN {X 0,Y 559.158,Z 280.827,A -85,B 0,C 180,E1 -2897.557,E2 -2897.557} C_VEL
LIN {X 0,Y 559.166,Z 280.826,A -85,B 0,C 180,E1 -2899.838,E2 -2899.838} C_VEL
LIN {X 0,Y 559.14,Z 280.831,A -85,B 0,C 180,E1 -2902.153,E2 -2902.153} C_VEL
LIN {X 0,Y 559.176,Z 280.828,A -85,B 0,C 180,E1 -2905.298,E2 -2905.298} C_VEL
LIN {X 0,Y 559.157,Z 280.827,A -85,B 0,C 180,E1 -2907.714,E2 -2907.714} C_VEL
LIN {X 0,Y 559.153,Z 280.829,A -85,B 0,C 180,E1 -2910.183,E2 -2910.183} C_VEL
LIN {X 0,Y 559.157,Z 280.832,A -85,B 0,C 180,E1 -2912.715,E2 -2912.715} C_VEL
LIN {X 0,Y 559.128,Z 280.837,A -85,B 0,C 180,E1 -2915.324,E2 -2915.324} C_VEL
LIN {X 0,Y 559.134,Z 280.831,A -85,B 0,C 180,E1 -2918.018,E2 -2918.018} C_VEL
LIN {X 0,Y 559.156,Z 280.827,A -85,B 0,C 180,E1 -2920.813,E2 -2920.813} C_VEL
LIN {X 0,Y 559.139,Z 280.834,A -85,B 0,C 180,E1 -2923.734,E2 -2923.734} C_VEL
LIN {X 0,Y 559.146,Z 280.83,A -85,B 0,C 180,E1 -2926.804,E2 -2926.804} C_VEL
LIN {X 0,Y 559.157,Z 280.832,A -85,B 0,C 180,E1 -2929.188,E2 -2929.188} C_VEL
LIN {X 0,Y 559.134,Z 280.834,A -85,B 0,C 180,E1 -2931.983,E2 -2931.983} C_VEL
LIN {X 0,Y 559.132,Z 280.831,A -85,B 0,C 180,E1 -2934.788,E2 -2934.788} C_VEL
LIN {X 0,Y 559.156,Z 280.832,A -85,B 0,C 180,E1 -2937.365,E2 -2937.365} C_VEL
LIN {X 0,Y 559.151,Z 280.836,A -85,B 0,C 180,E1 -2940.143,E2 -2940.143} C_VEL
LIN {X 0,Y 559.166,Z 280.828,A -85,B 0,C 180,E1 -2943.097,E2 -2943.097} C_VEL
LIN {X 0,Y 559.184,Z 280.835,A -85,B 0,C 180,E1 -2946.088,E2 -2946.088} C_VEL
LIN {X 0,Y 559.188,Z 280.979,A -85,B 0,C 180,E1 -2946.261,E2 -2946.261} C_VEL
LIN {X 0,Y 560.099,Z 286.478,A -85,B 0,C 180,E1 -2947.109,E2 -2947.109} C_VEL
LIN {X 0,Y 559.892,Z 306.293,A -85,B 0,C 180,E1 -2949.998,E2 -2949.998} C_VEL
LIN {X 0,Y 559.625,Z 326.669,A -85,B 0,C 180,E1 -2952.924,E2 -2952.924} C_VEL
LIN {X 0,Y 559.396,Z 346.612,A -85,B 0,C 180,E1 -2955.795,E2 -2955.795} C_VEL
LIN {X 0,Y 560.279,Z 354.286,A -85,B 0,C 180,E1 -2955.934,E2 -2955.934} C_VEL
LIN {X 0,Y 560.037,Z 454.939,A -85,B 0,C 180,E1 -2957.245,E2 -2957.245} C_VEL
LIN {X 0,Y 559.915,Z 468.212,A -85,B 0,C 180,E1 -2957.564,E2 -2957.564} C_VEL
LIN {X 0,Y 559.797,Z 480.374,A -85,B 0,C 180,E1 -2957.999,E2 -2957.999} C_VEL
LIN {X 0,Y 559.669,Z 491.807,A -85,B 0,C 180,E1 -2958.547,E2 -2958.547} C_VEL
LIN {X 0,Y 559.505,Z 502.902,A -85,B 0,C 180,E1 -2959.231,E2 -2959.231} C_VEL
LIN {X 0,Y 559.309,Z 513.536,A -85,B 0,C 180,E1 -2960.051,E2 -2960.051} C_VEL
LIN {X 0,Y 559.161,Z 523.095,A -85,B 0,C 180,E1 -2960.961,E2 -2960.961} C_VEL
LIN {X 0,Y 559.047,Z 530.959,A -85,B 0,C 180,E1 -2961.869,E2 -2961.869} C_VEL
LIN {X 0,Y 558.944,Z 538.621,A -85,B 0,C 180,E1 -2962.958,E2 -2962.958} C_VEL
LIN {X 0,Y 558.936,Z 545.679,A -85,B 0,C 180,E1 -2964.227,E2 -2964.227} C_VEL
LIN {X 0,Y 558.826,Z 550.372,A -85,B 0,C 180,E1 -2965.311,E2 -2965.311} C_VEL
LIN {X 0,Y 558.836,Z 553.957,A -85,B 0,C 180,E1 -2966.395,E2 -2966.395} C_VEL
LIN {X 0,Y 558.799,Z 555.807,A -85,B 0,C 180,E1 -2967.116,E2 -2967.116} C_VEL
LIN {X 0,Y 558.745,Z 558.184,A -85,B 0,C 180,E1 -2968.558,E2 -2968.558} C_VEL
LIN {X 0,Y 558.74,Z 559,A -85,B 0,C 180,E1 -2970,E2 -2970} C_VEL
LIN {X 0,Y 558.745,Z 558.185,A -85,B 0,C 180,E1 -2971.441,E2 -2971.441} C_VEL
LIN {X 0,Y 558.799,Z 555.811,A -85,B 0,C 180,E1 -2972.883,E2 -2972.883} C_VEL
LIN {X 0,Y 558.843,Z 552.896,A -85,B 0,C 180,E1 -2973.966,E2 -2973.966} C_VEL
LIN {X 0,Y 558.798,Z 548.95,A -85,B 0,C 180,E1 -2975.05,E2 -2975.05} C_VEL
LIN {X 0,Y 558.92,Z 543.869,A -85,B 0,C 180,E1 -2976.135,E2 -2976.135} C_VEL
LIN {X 0,Y 558.977,Z 537.47,A -85,B 0,C 180,E1 -2977.223,E2 -2977.223} C_VEL
LIN {X 0,Y 559.091,Z 529.48,A -85,B 0,C 180,E1 -2978.311,E2 -2978.311} C_VEL
LIN {X 0,Y 559.184,Z 521.337,A -85,B 0,C 180,E1 -2979.221,E2 -2979.221} C_VEL
LIN {X 0,Y 559.347,Z 511.403,A -85,B 0,C 180,E1 -2980.131,E2 -2980.131} C_VEL
LIN {X 0,Y 559.57,Z 500.385,A -85,B 0,C 180,E1 -2980.937,E2 -2980.937} C_VEL
LIN {X 0,Y 559.671,Z 488.466,A -85,B 0,C 180,E1 -2981.627,E2 -2981.627} C_VEL
LIN {X 0,Y 559.813,Z 475.778,A -85,B 0,C 180,E1 -2982.184,E2 -2982.184} C_VEL
LIN {X 0,Y 559.927,Z 462.36,A -85,B 0,C 180,E1 -2982.596,E2 -2982.596} C_VEL
LIN {X 0,Y 560.097,Z 449.111,A -85,B 0,C 180,E1 -2982.846,E2 -2982.846} C_VEL
LIN {X 0,Y 560.223,Z 352.314,A -85,B 0,C 180,E1 -2984.093,E2 -2984.093} C_VEL
LIN {X 0,Y 559.409,Z 346.616,A -85,B 0,C 180,E1 -2984.204,E2 -2984.204} C_VEL
LIN {X 0,Y 559.618,Z 324.696,A -85,B 0,C 180,E1 -2987.359,E2 -2987.359} C_VEL
LIN {X 0,Y 559.897,Z 305.022,A -85,B 0,C 180,E1 -2990.193,E2 -2990.193} C_VEL
LIN {X 0,Y 560.143,Z 286.589,A -85,B 0,C 180,E1 -2992.889,E2 -2992.889} C_VEL
LIN {X 0,Y 559.187,Z 280.835,A -85,B 0,C 180,E1 -2993.813,E2 -2993.813} C_VEL
LIN {X 0,Y 559.171,Z 280.827,A -85,B 0,C 180,E1 -2996.827,E2 -2996.827} C_VEL
LIN {X 0,Y 559.142,Z 280.832,A -85,B 0,C 180,E1 -2999.353,E2 -2999.353} C_VEL
LIN {X 0,Y 559.165,Z 280.832,A -85,B 0,C 180,E1 -3001.862,E2 -3001.862} C_VEL
LIN {X 0,Y 559.143,Z 280.836,A -85,B 0,C 180,E1 -3004.444,E2 -3004.444} C_VEL
LIN {X 0,Y 559.14,Z 280.83,A -85,B 0,C 180,E1 -3007.108,E2 -3007.108} C_VEL
LIN {X 0,Y 559.159,Z 280.831,A -85,B 0,C 180,E1 -3009.941,E2 -3009.941} C_VEL
LIN {X 0,Y 559.16,Z 280.832,A -85,B 0,C 180,E1 -3012.743,E2 -3012.743} C_VEL
LIN {X 0,Y 559.148,Z 280.829,A -85,B 0,C 180,E1 -3015.76,E2 -3015.76} C_VEL
LIN {X 0,Y 559.187,Z 280.828,A -85,B 0,C 180,E1 -3018.232,E2 -3018.232} C_VEL
LIN {X 0,Y 559.172,Z 280.828,A -85,B 0,C 180,E1 -3021.191,E2 -3021.191} C_VEL
LIN {X 0,Y 559.137,Z 280.83,A -85,B 0,C 180,E1 -3023.789,E2 -3023.789} C_VEL
LIN {X 0,Y 559.159,Z 280.831,A -85,B 0,C 180,E1 -3026.425,E2 -3026.425} C_VEL
LIN {X 0,Y 559.16,Z 280.836,A -85,B 0,C 180,E1 -3028.981,E2 -3028.981} C_VEL
LIN {X 0,Y 559.164,Z 280.828,A -85,B 0,C 180,E1 -3031.618,E2 -3031.618} C_VEL
LIN {X 0,Y 559.178,Z 280.825,A -85,B 0,C 180,E1 -3033.903,E2 -3033.903} C_VEL
LIN {X 0,Y 559.152,Z 280.831,A -85,B 0,C 180,E1 -3036.567,E2 -3036.567} C_VEL
LIN {X 0,Y 559.175,Z 280.832,A -85,B 0,C 180,E1 -3039.395,E2 -3039.395} C_VEL
LIN {X 0,Y 559.141,Z 280.833,A -85,B 0,C 180,E1 -3041.685,E2 -3041.685} C_VEL
LIN {X 0,Y 559.161,Z 280.828,A -85,B 0,C 180,E1 -3043.948,E2 -3043.948} C_VEL
LIN {X 0,Y 559.167,Z 280.826,A -85,B 0,C 180,E1 -3046.184,E2 -3046.184} C_VEL
LIN {X 0,Y 559.189,Z 280.829,A -85,B 0,C 180,E1 -3049.133,E2 -3049.133} C_VEL
LIN {X 0,Y 559.2,Z 280.824,A -85,B 0,C 180,E1 -3052.053,E2 -3052.053} C_VEL
LIN {X 0,Y 559.25,Z 280.817,A -85,B 0,C 180,E1 -3054.953,E2 -3054.953} C_VEL
LIN {X 0,Y 559.241,Z 280.825,A -85,B 0,C 180,E1 -3057.839,E2 -3057.839} C_VEL
LIN {X 0,Y 559.263,Z 280.814,A -85,B 0,C 180,E1 -3060.72,E2 -3060.72} C_VEL
LIN {X 0,Y 559.231,Z 280.818,A -85,B 0,C 180,E1 -3062.881,E2 -3062.881} C_VEL
LIN {X 0,Y 559.223,Z 280.828,A -85,B 0,C 180,E1 -3065.77,E2 -3065.77} C_VEL
LIN {X 0,Y 559.18,Z 280.825,A -85,B 0,C 180,E1 -3068.674,E2 -3068.674} C_VEL
LIN {X 0,Y 559.199,Z 280.826,A -85,B 0,C 180,E1 -3071.6,E2 -3071.6} C_VEL
LIN {X 0,Y 559.174,Z 280.828,A -85,B 0,C 180,E1 -3074.588,E2 -3074.588} C_VEL
LIN {X 0,Y 559.135,Z 280.832,A -85,B 0,C 180,E1 -3077.558,E2 -3077.558} C_VEL
LIN {X 0,Y 559.16,Z 280.831,A -85,B 0,C 180,E1 -3079.838,E2 -3079.838} C_VEL
LIN {X 0,Y 559.134,Z 280.838,A -85,B 0,C 180,E1 -3082.153,E2 -3082.153} C_VEL
LIN {X 0,Y 559.17,Z 280.826,A -85,B 0,C 180,E1 -3085.298,E2 -3085.298} C_VEL
LIN {X 0,Y 559.162,Z 280.835,A -85,B 0,C 180,E1 -3088.381,E2 -3088.381} C_VEL
LIN {X 0,Y 559.132,Z 280.833,A -85,B 0,C 180,E1 -3090.6,E2 -3090.6} C_VEL
LIN {X 0,Y 558.469,Z 280.916,A -85,B 0,C 180,E1 -3091.201,E2 -3091.201} C_VEL
LIN {X 0,Y 555.606,Z 281.273,A -85,B 0,C 180,E1 -3092.177,E2 -3092.177} C_VEL
LIN {X 0,Y 553.195,Z 281.575,A -85,B 0,C 180,E1 -3092.963,E2 -3092.963} C_VEL
LIN {X 0,Y 552.176,Z 281.698,A -85,B 0,C 180,E1 -3093.569,E2 -3093.569} C_VEL
LIN {X 0,Y 552.102,Z 281.706,A -85,B 0,C 180,E1 -3093.775,E2 -3093.775} C_VEL
LIN {X 0,Y 552.099,Z 281.717,A -85,B 0,C 180,E1 -3096.747,E2 -3096.747} C_VEL
LIN {X 0,Y 552.122,Z 281.705,A -85,B 0,C 180,E1 -3099.528,E2 -3099.528} C_VEL
LIN {X 0,Y 552.125,Z 281.707,A -85,B 0,C 180,E1 -3102.426,E2 -3102.426} C_VEL
LIN {X 0,Y 552.088,Z 281.71,A -85,B 0,C 180,E1 -3105.563,E2 -3105.563} C_VEL
LIN {X 0,Y 552.071,Z 281.713,A -85,B 0,C 180,E1 -3108.55,E2 -3108.55} C_VEL
LIN {X 0,Y 552.11,Z 281.711,A -85,B 0,C 180,E1 -3111.411,E2 -3111.411} C_VEL
LIN {X 0,Y 552.081,Z 281.709,A -85,B 0,C 180,E1 -3114.157,E2 -3114.157} C_VEL
LIN {X 0,Y 552.101,Z 281.71,A -85,B 0,C 180,E1 -3116.814,E2 -3116.814} C_VEL
LIN {X 0,Y 552.085,Z 281.718,A -85,B 0,C 180,E1 -3119.39,E2 -3119.39} C_VEL
LIN {X 0,Y 552.072,Z 281.713,A -85,B 0,C 180,E1 -3121.9,E2 -3121.9} C_VEL
LIN {X 0,Y 552.078,Z 281.71,A -85,B 0,C 180,E1 -3124.667,E2 -3124.667} C_VEL
LIN {X 0,Y 552.087,Z 281.719,A -85,B 0,C 180,E1 -3127.549,E2 -3127.549} C_VEL
LIN {X 0,Y 552.143,Z 281.702,A -85,B 0,C 180,E1 -3130.376,E2 -3130.376} C_VEL
LIN {X 0,Y 552.105,Z 281.707,A -85,B 0,C 180,E1 -3132.976,E2 -3132.976} C_VEL
LIN {X 0,Y 552.123,Z 281.711,A -85,B 0,C 180,E1 -3136.005,E2 -3136.005} C_VEL
LIN {X 0,Y 552.124,Z 281.706,A -85,B 0,C 180,E1 -3138.993,E2 -3138.993} C_VEL
LIN {X 0,Y 552.107,Z 281.72,A -85,B 0,C 180,E1 -3140.752,E2 -3140.752} C_VEL
LIN {X 0,Y 552.445,Z 287.253,A -85,B 0,C 180,E1 -3141.772,E2 -3141.772} C_VEL
LIN {X 0,Y 552.259,Z 302.269,A -85,B 0,C 180,E1 -3144.523,E2 -3144.523} C_VEL
LIN {X 0,Y 552.144,Z 308.489,A -85,B 0,C 180,E1 -3145.689,E2 -3145.689} C_VEL
LIN {X 0,Y 553.445,Z 316.943,A -85,B 0,C 180,E1 -3145.836,E2 -3145.836} C_VEL
LIN {X 0,Y 553.108,Z 415.202,A -85,B 0,C 180,E1 -3147.133,E2 -3147.133} C_VEL
LIN {X 0,Y 552.957,Z 428.22,A -85,B 0,C 180,E1 -3147.451,E2 -3147.451} C_VEL
LIN {X 0,Y 552.851,Z 440.729,A -85,B 0,C 180,E1 -3147.906,E2 -3147.906} C_VEL
LIN {X 0,Y 552.677,Z 451.933,A -85,B 0,C 180,E1 -3148.452,E2 -3148.452} C_VEL
LIN {X 0,Y 552.418,Z 463.513,A -85,B 0,C 180,E1 -3149.18,E2 -3149.18} C_VEL
LIN {X 0,Y 552.25,Z 473.916,A -85,B 0,C 180,E1 -3150,E2 -3150} C_VEL
LIN {X 0,Y 552.112,Z 483.323,A -85,B 0,C 180,E1 -3150.912,E2 -3150.912} C_VEL
LIN {X 0,Y 551.954,Z 492.432,A -85,B 0,C 180,E1 -3152.007,E2 -3152.007} C_VEL
LIN {X 0,Y 551.841,Z 499.781,A -85,B 0,C 180,E1 -3153.103,E2 -3153.103} C_VEL
LIN {X 0,Y 551.798,Z 506.57,A -85,B 0,C 180,E1 -3154.383,E2 -3154.383} C_VEL
LIN {X 0,Y 551.772,Z 511.066,A -85,B 0,C 180,E1 -3155.482,E2 -3155.482} C_VEL
LIN {X 0,Y 551.743,Z 514.495,A -85,B 0,C 180,E1 -3156.583,E2 -3156.583} C_VEL
LIN {X 0,Y 551.689,Z 516.203,A -85,B 0,C 180,E1 -3157.319,E2 -3157.319} C_VEL
LIN {X 0,Y 551.694,Z 517.505,A -85,B 0,C 180,E1 -3158.055,E2 -3158.055} C_VEL
LIN {X 0,Y 551.669,Z 518.411,A -85,B 0,C 180,E1 -3158.794,E2 -3158.794} C_VEL
LIN {X 0,Y 551.657,Z 518.895,A -85,B 0,C 180,E1 -3159.533,E2 -3159.533} C_VEL
LIN {X 0,Y 551.699,Z 518.627,A -85,B 0,C 180,E1 -3161.016,E2 -3161.016} C_VEL
LIN {X 0,Y 551.671,Z 517.901,A -85,B 0,C 180,E1 -3161.761,E2 -3161.761} C_VEL
LIN {X 0,Y 551.663,Z 516.722,A -85,B 0,C 180,E1 -3162.508,E2 -3162.508} C_VEL
LIN {X 0,Y 551.702,Z 514.149,A -85,B 0,C 180,E1 -3163.631,E2 -3163.631} C_VEL
LIN {X 0,Y 551.766,Z 510.51,A -85,B 0,C 180,E1 -3164.759,E2 -3164.759} C_VEL
LIN {X 0,Y 551.792,Z 505.681,A -85,B 0,C 180,E1 -3165.893,E2 -3165.893} C_VEL
LIN {X 0,Y 551.899,Z 499.509,A -85,B 0,C 180,E1 -3167.031,E2 -3167.031} C_VEL
LIN {X 0,Y 551.978,Z 491.743,A -85,B 0,C 180,E1 -3168.176,E2 -3168.176} C_VEL
LIN {X 0,Y 552.102,Z 483.725,A -85,B 0,C 180,E1 -3169.134,E2 -3169.134} C_VEL
LIN {X 0,Y 552.286,Z 473.844,A -85,B 0,C 180,E1 -3170.095,E2 -3170.095} C_VEL
LIN {X 0,Y 552.438,Z 462.735,A -85,B 0,C 180,E1 -3170.965,E2 -3170.965} C_VEL
LIN {X 0,Y 552.666,Z 451.894,A -85,B 0,C 180,E1 -3171.64,E2 -3171.64} C_VEL
LIN {X 0,Y 552.806,Z 439.195,A -85,B 0,C 180,E1 -3172.249,E2 -3172.249} C_VEL
LIN {X 0,Y 552.942,Z 425.917,A -85,B 0,C 180,E1 -3172.71,E2 -3172.71} C_VEL
LIN {X 0,Y 553.035,Z 414.23,A -85,B 0,C 180,E1 -3172.978,E2 -3172.978} C_VEL
LIN {X 0,Y 553.366,Z 315.675,A -85,B 0,C 180,E1 -3174.273,E2 -3174.273} C_VEL
LIN {X 0,Y 552.171,Z 308.398,A -85,B 0,C 180,E1 -3174.415,E2 -3174.415} C_VEL
LIN {X 0,Y 552.319,Z 295.695,A -85,B 0,C 180,E1 -3176.742,E2 -3176.742} C_VEL
LIN {X 0,Y 552.417,Z 283.614,A -85,B 0,C 180,E1 -3178.911,E2 -3178.911} C_VEL
LIN {X 0,Y 552.193,Z 281.703,A -85,B 0,C 180,E1 -3179.289,E2 -3179.289} C_VEL
LIN {X 0,Y 552.114,Z 281.715,A -85,B 0,C 180,E1 -3182.319,E2 -3182.319} C_VEL
LIN {X 0,Y 552.083,Z 281.712,A -85,B 0,C 180,E1 -3184.949,E2 -3184.949} C_VEL
LIN {X 0,Y 552.095,Z 281.708,A -85,B 0,C 180,E1 -3187.886,E2 -3187.886} C_VEL
LIN {X 0,Y 552.108,Z 281.716,A -85,B 0,C 180,E1 -3190.481,E2 -3190.481} C_VEL
LIN {X 0,Y 552.106,Z 281.707,A -85,B 0,C 180,E1 -3193.424,E2 -3193.424} C_VEL
LIN {X 0,Y 552.106,Z 281.715,A -85,B 0,C 180,E1 -3196.576,E2 -3196.576} C_VEL
LIN {X 0,Y 552.107,Z 281.707,A -85,B 0,C 180,E1 -3199.519,E2 -3199.519} C_VEL
LIN {X 0,Y 552.092,Z 281.709,A -85,B 0,C 180,E1 -3202.336,E2 -3202.336} C_VEL
LIN {X 0,Y 552.107,Z 281.714,A -85,B 0,C 180,E1 -3205.053,E2 -3205.053} C_VEL
LIN {X 0,Y 552.114,Z 281.705,A -85,B 0,C 180,E1 -3207.681,E2 -3207.681} C_VEL
LIN {X 0,Y 552.11,Z 281.704,A -85,B 0,C 180,E1 -3210.235,E2 -3210.235} C_VEL
LIN {X 0,Y 552.137,Z 281.707,A -85,B 0,C 180,E1 -3213,E2 -3213} C_VEL
LIN {X 0,Y 552.113,Z 281.713,A -85,B 0,C 180,E1 -3215.161,E2 -3215.161} C_VEL
LIN {X 0,Y 552.124,Z 281.703,A -85,B 0,C 180,E1 -3218.337,E2 -3218.337} C_VEL
LIN {X 0,Y 552.15,Z 281.699,A -85,B 0,C 180,E1 -3220.674,E2 -3220.674} C_VEL
LIN {X 0,Y 552.115,Z 281.71,A -85,B 0,C 180,E1 -3223.737,E2 -3223.737} C_VEL
LIN {X 0,Y 552.134,Z 281.707,A -85,B 0,C 180,E1 -3226.005,E2 -3226.005} C_VEL
LIN {X 0,Y 552.16,Z 281.699,A -85,B 0,C 180,E1 -3228.994,E2 -3228.994} C_VEL
LIN {X 0,Y 552.156,Z 281.707,A -85,B 0,C 180,E1 -3231.952,E2 -3231.952} C_VEL
LIN {X 0,Y 552.224,Z 281.691,A -85,B 0,C 180,E1 -3234.889,E2 -3234.889} C_VEL
LIN {X 0,Y 552.224,Z 281.699,A -85,B 0,C 180,E1 -3237.812,E2 -3237.812} C_VEL
LIN {X 0,Y 552.24,Z 281.69,A -85,B 0,C 180,E1 -3240.729,E2 -3240.729} C_VEL
LIN {X 0,Y 552.203,Z 281.693,A -85,B 0,C 180,E1 -3242.918,E2 -3242.918} C_VEL
LIN {X 0,Y 552.195,Z 281.699,A -85,B 0,C 180,E1 -3245.844,E2 -3245.844} C_VEL
LIN {X 0,Y 552.157,Z 281.702,A -85,B 0,C 180,E1 -3248.786,E2 -3248.786} C_VEL
LIN {X 0,Y 552.162,Z 281.698,A -85,B 0,C 180,E1 -3251.751,E2 -3251.751} C_VEL
LIN {X 0,Y 552.136,Z 281.707,A -85,B 0,C 180,E1 -3254.749,E2 -3254.749} C_VEL
LIN {X 0,Y 552.109,Z 281.706,A -85,B 0,C 180,E1 -3257.789,E2 -3257.789} C_VEL
LIN {X 0,Y 552.126,Z 281.705,A -85,B 0,C 180,E1 -3260.102,E2 -3260.102} C_VEL
LIN {X 0,Y 552.092,Z 281.713,A -85,B 0,C 180,E1 -3262.451,E2 -3262.451} C_VEL
LIN {X 0,Y 552.156,Z 281.702,A -85,B 0,C 180,E1 -3265.351,E2 -3265.351} C_VEL
LIN {X 0,Y 552.11,Z 281.705,A -85,B 0,C 180,E1 -3268.099,E2 -3268.099} C_VEL
LIN {X 0,Y 552.103,Z 281.711,A -85,B 0,C 180,E1 -3270.609,E2 -3270.609} C_VEL
LIN {X 0,Y 552.115,Z 281.713,A -85,B 0,C 180,E1 -3273.186,E2 -3273.186} C_VEL
LIN {X 0,Y 552.086,Z 281.708,A -85,B 0,C 180,E1 -3275.844,E2 -3275.844} C_VEL
LIN {X 0,Y 552.118,Z 281.706,A -85,B 0,C 180,E1 -3278.589,E2 -3278.589} C_VEL
LIN {X 0,Y 552.122,Z 281.712,A -85,B 0,C 180,E1 -3281.446,E2 -3281.446} C_VEL
LIN {X 0,Y 552.089,Z 281.708,A -85,B 0,C 180,E1 -3284.531,E2 -3284.531} C_VEL
LIN {X 0,Y 552.131,Z 281.713,A -85,B 0,C 180,E1 -3287.585,E2 -3287.585} C_VEL
LIN {X 0,Y 552.13,Z 281.703,A -85,B 0,C 180,E1 -3290.473,E2 -3290.473} C_VEL
LIN {X 0,Y 552.108,Z 281.709,A -85,B 0,C 180,E1 -3293.317,E2 -3293.317} C_VEL
LIN {X 0,Y 552.128,Z 281.712,A -85,B 0,C 180,E1 -3295.939,E2 -3295.939} C_VEL
LIN {X 0,Y 552.122,Z 281.706,A -85,B 0,C 180,E1 -3298.541,E2 -3298.541} C_VEL
LIN {X 0,Y 552.127,Z 281.708,A -85,B 0,C 180,E1 -3301.438,E2 -3301.438} C_VEL
LIN {X 0,Y 552.131,Z 281.711,A -85,B 0,C 180,E1 -3304.356,E2 -3304.356} C_VEL
LIN {X 0,Y 552.158,Z 281.843,A -85,B 0,C 180,E1 -3306.115,E2 -3306.115} C_VEL
LIN {X 0,Y 553.192,Z 288.838,A -85,B 0,C 180,E1 -3307.202,E2 -3307.202} C_VEL
LIN {X 0,Y 552.889,Z 308.911,A -85,B 0,C 180,E1 -3310.161,E2 -3310.161} C_VEL
LIN {X 0,Y 552.596,Z 328.389,A -85,B 0,C 180,E1 -3312.991,E2 -3312.991} C_VEL
LIN {X 0,Y 552.373,Z 346.706,A -85,B 0,C 180,E1 -3315.625,E2 -3315.625} C_VEL
LIN {X 0,Y 553.416,Z 354.774,A -85,B 0,C 180,E1 -3315.762,E2 -3315.762} C_VEL
LIN {X 0,Y 553.112,Z 454.939,A -85,B 0,C 180,E1 -3317.082,E2 -3317.082} C_VEL
LIN {X 0,Y 552.995,Z 468.212,A -85,B 0,C 180,E1 -3317.406,E2 -3317.406} C_VEL
LIN {X 0,Y 552.84,Z 480.365,A -85,B 0,C 180,E1 -3317.845,E2 -3317.845} C_VEL
LIN {X 0,Y 552.695,Z 492.622,A -85,B 0,C 180,E1 -3318.447,E2 -3318.447} C_VEL
LIN {X 0,Y 552.5,Z 504.192,A -85,B 0,C 180,E1 -3319.186,E2 -3319.186} C_VEL
LIN {X 0,Y 552.295,Z 514.604,A -85,B 0,C 180,E1 -3320.015,E2 -3320.015} C_VEL
LIN {X 0,Y 552.126,Z 523.108,A -85,B 0,C 180,E1 -3320.844,E2 -3320.844} C_VEL
LIN {X 0,Y 552.009,Z 530.959,A -85,B 0,C 180,E1 -3321.765,E2 -3321.765} C_VEL
LIN {X 0,Y 551.89,Z 538.62,A -85,B 0,C 180,E1 -3322.868,E2 -3322.868} C_VEL
LIN {X 0,Y 551.868,Z 545.678,A -85,B 0,C 180,E1 -3324.152,E2 -3324.152} C_VEL
LIN {X 0,Y 551.725,Z 550.372,A -85,B 0,C 180,E1 -3325.25,E2 -3325.25} C_VEL
LIN {X 0,Y 551.75,Z 553.958,A -85,B 0,C 180,E1 -3326.348,E2 -3326.348} C_VEL
LIN {X 0,Y 551.723,Z 555.807,A -85,B 0,C 180,E1 -3327.079,E2 -3327.079} C_VEL
LIN {X 0,Y 551.644,Z 558.183,A -85,B 0,C 180,E1 -3328.54,E2 -3328.54} C_VEL
LIN {X 0,Y 551.64,Z 559,A -85,B 0,C 180,E1 -3330,E2 -3330} C_VEL
LIN {X 0,Y 551.644,Z 558.185,A -85,B 0,C 180,E1 -3331.46,E2 -3331.46} C_VEL
LIN {X 0,Y 551.723,Z 555.811,A -85,B 0,C 180,E1 -3332.92,E2 -3332.92} C_VEL
LIN {X 0,Y 551.763,Z 552.896,A -85,B 0,C 180,E1 -3334.017,E2 -3334.017} C_VEL
LIN {X 0,Y 551.723,Z 548.949,A -85,B 0,C 180,E1 -3335.115,E2 -3335.115} C_VEL
LIN {X 0,Y 551.814,Z 543.127,A -85,B 0,C 180,E1 -3336.353,E2 -3336.353} C_VEL
LIN {X 0,Y 551.926,Z 536.238,A -85,B 0,C 180,E1 -3337.499,E2 -3337.499} C_VEL
LIN {X 0,Y 552.064,Z 527.994,A -85,B 0,C 180,E1 -3338.602,E2 -3338.602} C_VEL
LIN {X 0,Y 552.222,Z 519.543,A -85,B 0,C 180,E1 -3339.523,E2 -3339.523} C_VEL
LIN {X 0,Y 552.406,Z 509.097,A -85,B 0,C 180,E1 -3340.445,E2 -3340.445} C_VEL
LIN {X 0,Y 552.609,Z 498.195,A -85,B 0,C 180,E1 -3341.219,E2 -3341.219} C_VEL
LIN {X 0,Y 552.75,Z 487.412,A -85,B 0,C 180,E1 -3341.83,E2 -3341.83} C_VEL
LIN {X 0,Y 552.883,Z 475.774,A -85,B 0,C 180,E1 -3342.34,E2 -3342.34} C_VEL
LIN {X 0,Y 553.005,Z 462.359,A -85,B 0,C 180,E1 -3342.756,E2 -3342.756} C_VEL
LIN {X 0,Y 553.182,Z 449.111,A -85,B 0,C 180,E1 -3343.009,E2 -3343.009} C_VEL
LIN {X 0,Y 553.255,Z 352.358,A -85,B 0,C 180,E1 -3344.273,E2 -3344.273} C_VEL
LIN {X 0,Y 552.382,Z 346.659,A -85,B 0,C 180,E1 -3344.381,E2 -3344.381} C_VEL
LIN {X 0,Y 552.632,Z 325.143,A -85,B 0,C 180,E1 -3347.484,E2 -3347.484} C_VEL
LIN {X 0,Y 552.926,Z 304.765,A -85,B 0,C 180,E1 -3350.459,E2 -3350.459} C_VEL
LIN {X 0,Y 553.171,Z 287.661,A -85,B 0,C 180,E1 -3352.996,E2 -3352.996} C_VEL
LIN {X 0,Y 552.148,Z 281.711,A -85,B 0,C 180,E1 -3353.946,E2 -3353.946} C_VEL
LIN {X 0,Y 552.119,Z 281.708,A -85,B 0,C 180,E1 -3356.456,E2 -3356.456} C_VEL
LIN {X 0,Y 552.11,Z 281.707,A -85,B 0,C 180,E1 -3358.928,E2 -3358.928} C_VEL
LIN {X 0,Y 552.111,Z 281.706,A -85,B 0,C 180,E1 -3361.475,E2 -3361.475} C_VEL
LIN {X 0,Y 552.132,Z 281.713,A -85,B 0,C 180,E1 -3364.17,E2 -3364.17} C_VEL
LIN {X 0,Y 552.104,Z 281.709,A -85,B 0,C 180,E1 -3366.746,E2 -3366.746} C_VEL
LIN {X 0,Y 552.128,Z 281.703,A -85,B 0,C 180,E1 -3369.527,E2 -3369.527} C_VEL
LIN {X 0,Y 552.129,Z 281.714,A -85,B 0,C 180,E1 -3372.425,E2 -3372.425} C_VEL
LIN {X 0,Y 552.093,Z 281.707,A -85,B 0,C 180,E1 -3375.562,E2 -3375.562} C_VEL
LIN {X 0,Y 552.13,Z 281.713,A -85,B 0,C 180,E1 -3378.555,E2 -3378.555} C_VEL
LIN {X 0,Y 552.115,Z 281.705,A -85,B 0,C 180,E1 -3381.411,E2 -3381.411} C_VEL
LIN {X 0,Y 552.085,Z 281.71,A -85,B 0,C 180,E1 -3384.156,E2 -3384.156} C_VEL
LIN {X 0,Y 552.112,Z 281.716,A -85,B 0,C 180,E1 -3386.814,E2 -3386.814} C_VEL
LIN {X 0,Y 552.104,Z 281.709,A -85,B 0,C 180,E1 -3389.391,E2 -3389.391} C_VEL
LIN {X 0,Y 552.116,Z 281.705,A -85,B 0,C 180,E1 -3391.902,E2 -3391.902} C_VEL
LIN {X 0,Y 552.152,Z 281.704,A -85,B 0,C 180,E1 -3394.649,E2 -3394.649} C_VEL
LIN {X 0,Y 552.091,Z 281.711,A -85,B 0,C 180,E1 -3397.549,E2 -3397.549} C_VEL
LIN {X 0,Y 552.144,Z 281.701,A -85,B 0,C 180,E1 -3400.373,E2 -3400.373} C_VEL
LIN {X 0,Y 552.15,Z 281.706,A -85,B 0,C 180,E1 -3402.977,E2 -3402.977} C_VEL
LIN {X 0,Y 552.131,Z 281.704,A -85,B 0,C 180,E1 -3406.004,E2 -3406.004} C_VEL
LIN {X 0,Y 552.157,Z 281.703,A -85,B 0,C 180,E1 -3408.993,E2 -3408.993} C_VEL
LIN {X 0,Y 552.154,Z 281.703,A -85,B 0,C 180,E1 -3411.951,E2 -3411.951} C_VEL
LIN {X 0,Y 552.225,Z 281.692,A -85,B 0,C 180,E1 -3414.889,E2 -3414.889} C_VEL
LIN {X 0,Y 552.214,Z 281.7,A -85,B 0,C 180,E1 -3417.812,E2 -3417.812} C_VEL
LIN {X 0,Y 552.234,Z 281.69,A -85,B 0,C 180,E1 -3420.729,E2 -3420.729} C_VEL
LIN {X 0,Y 552.198,Z 281.694,A -85,B 0,C 180,E1 -3422.918,E2 -3422.918} C_VEL
LIN {X 0,Y 552.191,Z 281.705,A -85,B 0,C 180,E1 -3425.844,E2 -3425.844} C_VEL
LIN {X 0,Y 552.151,Z 281.7,A -85,B 0,C 180,E1 -3428.786,E2 -3428.786} C_VEL
LIN {X 0,Y 552.157,Z 281.705,A -85,B 0,C 180,E1 -3431.75,E2 -3431.75} C_VEL
LIN {X 0,Y 552.122,Z 281.705,A -85,B 0,C 180,E1 -3434.749,E2 -3434.749} C_VEL
LIN {X 0,Y 552.092,Z 281.711,A -85,B 0,C 180,E1 -3437.789,E2 -3437.789} C_VEL
LIN {X 0,Y 552.12,Z 281.712,A -85,B 0,C 180,E1 -3440.101,E2 -3440.101} C_VEL
LIN {X 0,Y 552.085,Z 281.717,A -85,B 0,C 180,E1 -3442.451,E2 -3442.451} C_VEL
LIN {X 0,Y 552.15,Z 281.7,A -85,B 0,C 180,E1 -3445.35,E2 -3445.35} C_VEL
LIN {X 0,Y 552.091,Z 281.712,A -85,B 0,C 180,E1 -3448.099,E2 -3448.099} C_VEL
LIN {X 0,Y 552.095,Z 281.717,A -85,B 0,C 180,E1 -3450.61,E2 -3450.61} C_VEL
LIN {X 0,Y 552.107,Z 281.708,A -85,B 0,C 180,E1 -3453.186,E2 -3453.186} C_VEL
LIN {X 0,Y 552.102,Z 281.706,A -85,B 0,C 180,E1 -3453.775,E2 -3453.775} C_VEL
LIN {X 0,Y 551.468,Z 281.792,A -85,B 0,C 180,E1 -3454.383,E2 -3454.383} C_VEL
LIN {X 0,Y 548.649,Z 282.148,A -85,B 0,C 180,E1 -3455.371,E2 -3455.371} C_VEL
LIN {X 0,Y 546.229,Z 282.451,A -85,B 0,C 180,E1 -3456.167,E2 -3456.167} C_VEL
LIN {X 0,Y 545.16,Z 282.581,A -85,B 0,C 180,E1 -3456.78,E2 -3456.78} C_VEL
LIN {X 0,Y 545.057,Z 282.59,A -85,B 0,C 180,E1 -3456.988,E2 -3456.988} C_VEL
LIN {X 0,Y 545.059,Z 282.585,A -85,B 0,C 180,E1 -3460.143,E2 -3460.143} C_VEL
LIN {X 0,Y 545.074,Z 282.589,A -85,B 0,C 180,E1 -3463.107,E2 -3463.107} C_VEL
LIN {X 0,Y 545.045,Z 282.586,A -85,B 0,C 180,E1 -3466.227,E2 -3466.227} C_VEL
LIN {X 0,Y 545.025,Z 282.595,A -85,B 0,C 180,E1 -3468.881,E2 -3468.881} C_VEL
LIN {X 0,Y 545.044,Z 282.587,A -85,B 0,C 180,E1 -3471.763,E2 -3471.763} C_VEL
LIN {X 0,Y 545.032,Z 282.588,A -85,B 0,C 180,E1 -3474.532,E2 -3474.532} C_VEL
LIN {X 0,Y 545.06,Z 282.593,A -85,B 0,C 180,E1 -3477.212,E2 -3477.212} C_VEL
LIN {X 0,Y 545.058,Z 282.587,A -85,B 0,C 180,E1 -3479.811,E2 -3479.811} C_VEL
LIN {X 0,Y 545.039,Z 282.586,A -85,B 0,C 180,E1 -3482.342,E2 -3482.342} C_VEL
LIN {X 0,Y 545.036,Z 282.588,A -85,B 0,C 180,E1 -3484.817,E2 -3484.817} C_VEL
LIN {X 0,Y 545.03,Z 282.592,A -85,B 0,C 180,E1 -3487.242,E2 -3487.242} C_VEL
LIN {X 0,Y 545.114,Z 282.577,A -85,B 0,C 180,E1 -3490.415,E2 -3490.415} C_VEL
LIN {X 0,Y 545.038,Z 282.593,A -85,B 0,C 180,E1 -3493.521,E2 -3493.521} C_VEL
LIN {X 0,Y 545.087,Z 282.591,A -85,B 0,C 180,E1 -3495.82,E2 -3495.82} C_VEL
LIN {X 0,Y 545.07,Z 282.585,A -85,B 0,C 180,E1 -3498.849,E2 -3498.849} C_VEL
LIN {X 0,Y 545.076,Z 282.609,A -85,B 0,C 180,E1 -3500.679,E2 -3500.679} C_VEL
LIN {X 0,Y 545.442,Z 287.878,A -85,B 0,C 180,E1 -3501.666,E2 -3501.666} C_VEL
LIN {X 0,Y 545.232,Z 304.065,A -85,B 0,C 180,E1 -3504.638,E2 -3504.638} C_VEL
LIN {X 0,Y 545.128,Z 308.603,A -85,B 0,C 180,E1 -3505.494,E2 -3505.494} C_VEL
LIN {X 0,Y 546.508,Z 316.646,A -85,B 0,C 180,E1 -3505.644,E2 -3505.644} C_VEL
LIN {X 0,Y 546.203,Z 414.995,A -85,B 0,C 180,E1 -3506.958,E2 -3506.958} C_VEL
LIN {X 0,Y 546.043,Z 428.144,A -85,B 0,C 180,E1 -3507.28,E2 -3507.28} C_VEL
LIN {X 0,Y 545.915,Z 440.705,A -85,B 0,C 180,E1 -3507.741,E2 -3507.741} C_VEL
LIN {X 0,Y 545.711,Z 452.733,A -85,B 0,C 180,E1 -3508.34,E2 -3508.34} C_VEL
LIN {X 0,Y 545.415,Z 464.151,A -85,B 0,C 180,E1 -3509.077,E2 -3509.077} C_VEL
LIN {X 0,Y 545.229,Z 474.421,A -85,B 0,C 180,E1 -3509.908,E2 -3509.908} C_VEL
LIN {X 0,Y 545.08,Z 482.843,A -85,B 0,C 180,E1 -3510.739,E2 -3510.739} C_VEL
LIN {X 0,Y 544.909,Z 492.038,A -85,B 0,C 180,E1 -3511.848,E2 -3511.848} C_VEL
LIN {X 0,Y 544.771,Z 499.455,A -85,B 0,C 180,E1 -3512.958,E2 -3512.958} C_VEL
LIN {X 0,Y 544.729,Z 505.429,A -85,B 0,C 180,E1 -3514.069,E2 -3514.069} C_VEL
LIN {X 0,Y 544.648,Z 510.176,A -85,B 0,C 180,E1 -3515.183,E2 -3515.183} C_VEL
LIN {X 0,Y 544.673,Z 514.436,A -85,B 0,C 180,E1 -3516.515,E2 -3516.515} C_VEL
LIN {X 0,Y 544.602,Z 516.46,A -85,B 0,C 180,E1 -3517.415,E2 -3517.415} C_VEL
LIN {X 0,Y 544.609,Z 517.704,A -85,B 0,C 180,E1 -3518.161,E2 -3518.161} C_VEL
LIN {X 0,Y 544.562,Z 518.529,A -85,B 0,C 180,E1 -3518.909,E2 -3518.909} C_VEL
LIN {X 0,Y 544.58,Z 518.923,A -85,B 0,C 180,E1 -3519.658,E2 -3519.658} C_VEL
LIN {X 0,Y 544.605,Z 518.54,A -85,B 0,C 180,E1 -3521.161,E2 -3521.161} C_VEL
LIN {X 0,Y 544.565,Z 517.72,A -85,B 0,C 180,E1 -3521.917,E2 -3521.917} C_VEL
LIN {X 0,Y 544.575,Z 516.46,A -85,B 0,C 180,E1 -3522.674,E2 -3522.674} C_VEL
LIN {X 0,Y 544.632,Z 513.765,A -85,B 0,C 180,E1 -3523.812,E2 -3523.812} C_VEL
LIN {X 0,Y 544.687,Z 509.993,A -85,B 0,C 180,E1 -3524.955,E2 -3524.955} C_VEL
LIN {X 0,Y 544.729,Z 505.021,A -85,B 0,C 180,E1 -3526.105,E2 -3526.105} C_VEL
LIN {X 0,Y 544.836,Z 498.194,A -85,B 0,C 180,E1 -3527.341,E2 -3527.341} C_VEL
LIN {X 0,Y 544.996,Z 490.715,A -85,B 0,C 180,E1 -3528.418,E2 -3528.418} C_VEL
LIN {X 0,Y 545.08,Z 482.467,A -85,B 0,C 180,E1 -3529.391,E2 -3529.391} C_VEL
LIN {X 0,Y 545.302,Z 472.343,A -85,B 0,C 180,E1 -3530.364,E2 -3530.364} C_VEL
LIN {X 0,Y 545.483,Z 462.303,A -85,B 0,C 180,E1 -3531.146,E2 -3531.146} C_VEL
LIN {X 0,Y 545.747,Z 451.313,A -85,B 0,C 180,E1 -3531.83,E2 -3531.83} C_VEL
LIN {X 0,Y 545.88,Z 438.43,A -85,B 0,C 180,E1 -3532.446,E2 -3532.446} C_VEL
LIN {X 0,Y 546.013,Z 425.576,A -85,B 0,C 180,E1 -3532.89,E2 -3532.89} C_VEL
LIN {X 0,Y 546.132,Z 413.466,A -85,B 0,C 180,E1 -3533.16,E2 -3533.16} C_VEL
LIN {X 0,Y 546.506,Z 316.435,A -85,B 0,C 180,E1 -3534.448,E2 -3534.448} C_VEL
LIN {X 0,Y 545.145,Z 308.548,A -85,B 0,C 180,E1 -3534.599,E2 -3534.599} C_VEL
LIN {X 0,Y 545.247,Z 298.653,A -85,B 0,C 180,E1 -3536.404,E2 -3536.404} C_VEL
LIN {X 0,Y 545.404,Z 285.432,A -85,B 0,C 180,E1 -3538.808,E2 -3538.808} C_VEL
LIN {X 0,Y 545.118,Z 282.585,A -85,B 0,C 180,E1 -3539.335,E2 -3539.335} C_VEL
LIN {X 0,Y 545.055,Z 282.592,A -85,B 0,C 180,E1 -3541.915,E2 -3541.915} C_VEL
LIN {X 0,Y 545.061,Z 282.591,A -85,B 0,C 180,E1 -3544.564,E2 -3544.564} C_VEL
LIN {X 0,Y 545.035,Z 282.586,A -85,B 0,C 180,E1 -3547.304,E2 -3547.304} C_VEL
LIN {X 0,Y 545.064,Z 282.589,A -85,B 0,C 180,E1 -3550.143,E2 -3550.143} C_VEL
LIN {X 0,Y 545.078,Z 282.585,A -85,B 0,C 180,E1 -3553.107,E2 -3553.107} C_VEL
LIN {X 0,Y 545.048,Z 282.589,A -85,B 0,C 180,E1 -3556.226,E2 -3556.226} C_VEL
LIN {X 0,Y 545.081,Z 282.59,A -85,B 0,C 180,E1 -3558.885,E2 -3558.885} C_VEL
LIN {X 0,Y 545.08,Z 282.591,A -85,B 0,C 180,E1 -3560.818,E2 -3560.818} C_VEL
LIN {X 0,Y 545.041,Z 282.586,A -85,B 0,C 180,E1 -3563.62,E2 -3563.62} C_VEL
LIN {X 0,Y 545.065,Z 282.583,A -85,B 0,C 180,E1 -3566.328,E2 -3566.328} C_VEL
LIN {X 0,Y 545.065,Z 282.59,A -85,B 0,C 180,E1 -3568.952,E2 -3568.952} C_VEL
LIN {X 0,Y 545.1,Z 282.581,A -85,B 0,C 180,E1 -3571.508,E2 -3571.508} C_VEL
LIN {X 0,Y 545.094,Z 282.579,A -85,B 0,C 180,E1 -3574.491,E2 -3574.491} C_VEL
LIN {X 0,Y 545.037,Z 282.593,A -85,B 0,C 180,E1 -3577.242,E2 -3577.242} C_VEL
LIN {X 0,Y 545.115,Z 282.575,A -85,B 0,C 180,E1 -3580.415,E2 -3580.415} C_VEL
LIN {X 0,Y 545.073,Z 282.592,A -85,B 0,C 180,E1 -3583.521,E2 -3583.521} C_VEL
LIN {X 0,Y 545.094,Z 282.586,A -85,B 0,C 180,E1 -3585.82,E2 -3585.82} C_VEL
LIN {X 0,Y 545.116,Z 282.576,A -85,B 0,C 180,E1 -3588.849,E2 -3588.849} C_VEL
LIN {X 0,Y 545.127,Z 282.584,A -85,B 0,C 180,E1 -3591.847,E2 -3591.847} C_VEL
LIN {X 0,Y 545.2,Z 282.566,A -85,B 0,C 180,E1 -3594.823,E2 -3594.823} C_VEL
LIN {X 0,Y 545.195,Z 282.574,A -85,B 0,C 180,E1 -3597.784,E2 -3597.784} C_VEL
LIN {X 0,Y 545.21,Z 282.566,A -85,B 0,C 180,E1 -3600.739,E2 -3600.739} C_VEL
LIN {X 0,Y 545.17,Z 282.569,A -85,B 0,C 180,E1 -3602.956,E2 -3602.956} C_VEL
LIN {X 0,Y 545.167,Z 282.575,A -85,B 0,C 180,E1 -3605.92,E2 -3605.92} C_VEL
LIN {X 0,Y 545.116,Z 282.578,A -85,B 0,C 180,E1 -3608.9,E2 -3608.9} C_VEL
LIN {X 0,Y 545.135,Z 282.575,A -85,B 0,C 180,E1 -3611.904,E2 -3611.904} C_VEL
LIN {X 0,Y 545.085,Z 282.583,A -85,B 0,C 180,E1 -3614.944,E2 -3614.944} C_VEL
LIN {X 0,Y 545.077,Z 282.583,A -85,B 0,C 180,E1 -3618.026,E2 -3618.026} C_VEL
LIN {X 0,Y 545.092,Z 282.584,A -85,B 0,C 180,E1 -3620.372,E2 -3620.372} C_VEL
LIN {X 0,Y 545.082,Z 282.581,A -85,B 0,C 180,E1 -3623.559,E2 -3623.559} C_VEL
LIN {X 0,Y 545.08,Z 282.581,A -85,B 0,C 180,E1 -3626.001,E2 -3626.001} C_VEL
LIN {X 0,Y 545.089,Z 282.587,A -85,B 0,C 180,E1 -3628.748,E2 -3628.748} C_VEL
LIN {X 0,Y 545.058,Z 282.584,A -85,B 0,C 180,E1 -3631.679,E2 -3631.679} C_VEL
LIN {X 0,Y 545.063,Z 282.586,A -85,B 0,C 180,E1 -3634.565,E2 -3634.565} C_VEL
LIN {X 0,Y 545.038,Z 282.595,A -85,B 0,C 180,E1 -3637.304,E2 -3637.304} C_VEL
LIN {X 0,Y 545.066,Z 282.579,A -85,B 0,C 180,E1 -3640.143,E2 -3640.143} C_VEL
LIN {X 0,Y 545.079,Z 282.587,A -85,B 0,C 180,E1 -3643.107,E2 -3643.107} C_VEL
LIN {X 0,Y 545.05,Z 282.586,A -85,B 0,C 180,E1 -3646.227,E2 -3646.227} C_VEL
LIN {X 0,Y 545.083,Z 282.583,A -85,B 0,C 180,E1 -3648.886,E2 -3648.886} C_VEL
LIN {X 0,Y 545.053,Z 282.592,A -85,B 0,C 180,E1 -3651.763,E2 -3651.763} C_VEL
LIN {X 0,Y 545.037,Z 282.588,A -85,B 0,C 180,E1 -3654.532,E2 -3654.532} C_VEL
LIN {X 0,Y 545.068,Z 282.586,A -85,B 0,C 180,E1 -3657.212,E2 -3657.212} C_VEL
LIN {X 0,Y 545.066,Z 282.592,A -85,B 0,C 180,E1 -3659.811,E2 -3659.811} C_VEL
LIN {X 0,Y 545.077,Z 282.587,A -85,B 0,C 180,E1 -3662.344,E2 -3662.344} C_VEL
LIN {X 0,Y 545.109,Z 282.582,A -85,B 0,C 180,E1 -3664.82,E2 -3664.82} C_VEL
LIN {X 0,Y 545.13,Z 282.717,A -85,B 0,C 180,E1 -3665.967,E2 -3665.967} C_VEL
LIN {X 0,Y 546.258,Z 289.868,A -85,B 0,C 180,E1 -3667.096,E2 -3667.096} C_VEL
LIN {X 0,Y 545.907,Z 310.201,A -85,B 0,C 180,E1 -3670.13,E2 -3670.13} C_VEL
LIN {X 0,Y 545.575,Z 329.424,A -85,B 0,C 180,E1 -3672.959,E2 -3672.959} C_VEL
LIN {X 0,Y 545.395,Z 346.73,A -85,B 0,C 180,E1 -3675.445,E2 -3675.445} C_VEL
LIN {X 0,Y 546.533,Z 355.307,A -85,B 0,C 180,E1 -3675.59,E2 -3675.59} C_VEL
LIN {X 0,Y 546.211,Z 454.799,A -85,B 0,C 180,E1 -3676.916,E2 -3676.916} C_VEL
LIN {X 0,Y 546.06,Z 468.1,A -85,B 0,C 180,E1 -3677.243,E2 -3677.243} C_VEL
LIN {X 0,Y 545.886,Z 480.285,A -85,B 0,C 180,E1 -3677.688,E2 -3677.688} C_VEL
LIN {X 0,Y 545.736,Z 492.587,A -85,B 0,C 180,E1 -3678.298,E2 -3678.298} C_VEL
LIN {X 0,Y 545.522,Z 504.189,A -85,B 0,C 180,E1 -3679.046,E2 -3679.046} C_VEL
LIN {X 0,Y 545.282,Z 514.602,A -85,B 0,C 180,E1 -3679.886,E2 -3679.886} C_VEL
LIN {X 0,Y 545.085,Z 523.112,A -85,B 0,C 180,E1 -3680.725,E2 -3680.725} C_VEL
LIN {X 0,Y 544.972,Z 530.959,A -85,B 0,C 180,E1 -3681.658,E2 -3681.658} C_VEL
LIN {X 0,Y 544.824,Z 538.62,A -85,B 0,C 180,E1 -3682.775,E2 -3682.775} C_VEL
LIN {X 0,Y 544.779,Z 545.678,A -85,B 0,C 180,E1 -3684.076,E2 -3684.076} C_VEL
LIN {X 0,Y 544.629,Z 550.372,A -85,B 0,C 180,E1 -3685.188,E2 -3685.188} C_VEL
LIN {X 0,Y 544.669,Z 553.957,A -85,B 0,C 180,E1 -3686.301,E2 -3686.301} C_VEL
LIN {X 0,Y 544.65,Z 555.806,A -85,B 0,C 180,E1 -3687.041,E2 -3687.041} C_VEL
LIN {X 0,Y 544.545,Z 558.182,A -85,B 0,C 180,E1 -3688.521,E2 -3688.521} C_VEL
LIN {X 0,Y 544.541,Z 559,A -85,B 0,C 180,E1 -3690,E2 -3690} C_VEL
LIN {X 0,Y 544.545,Z 558.184,A -85,B 0,C 180,E1 -3691.479,E2 -3691.479} C_VEL
LIN {X 0,Y 544.65,Z 555.811,A -85,B 0,C 180,E1 -3692.958,E2 -3692.958} C_VEL
LIN {X 0,Y 544.683,Z 552.896,A -85,B 0,C 180,E1 -3694.069,E2 -3694.069} C_VEL
LIN {X 0,Y 544.653,Z 548.949,A -85,B 0,C 180,E1 -3695.182,E2 -3695.182} C_VEL
LIN {X 0,Y 544.729,Z 543.646,A -85,B 0,C 180,E1 -3696.339,E2 -3696.339} C_VEL
LIN {X 0,Y 544.859,Z 536.237,A -85,B 0,C 180,E1 -3697.597,E2 -3697.597} C_VEL
LIN {X 0,Y 545.016,Z 527.995,A -85,B 0,C 180,E1 -3698.714,E2 -3698.714} C_VEL
LIN {X 0,Y 545.202,Z 519.543,A -85,B 0,C 180,E1 -3699.647,E2 -3699.647} C_VEL
LIN {X 0,Y 545.387,Z 509.095,A -85,B 0,C 180,E1 -3700.581,E2 -3700.581} C_VEL
LIN {X 0,Y 545.624,Z 497.384,A -85,B 0,C 180,E1 -3701.417,E2 -3701.417} C_VEL
LIN {X 0,Y 545.82,Z 485.433,A -85,B 0,C 180,E1 -3702.077,E2 -3702.077} C_VEL
LIN {X 0,Y 545.981,Z 473.077,A -85,B 0,C 180,E1 -3702.593,E2 -3702.593} C_VEL
LIN {X 0,Y 546.141,Z 460.404,A -85,B 0,C 180,E1 -3702.967,E2 -3702.967} C_VEL
LIN {X 0,Y 546.259,Z 447.19,A -85,B 0,C 180,E1 -3703.201,E2 -3703.201} C_VEL
LIN {X 0,Y 546.451,Z 353.598,A -85,B 0,C 180,E1 -3704.435,E2 -3704.435} C_VEL
LIN {X 0,Y 545.358,Z 346.416,A -85,B 0,C 180,E1 -3704.569,E2 -3704.569} C_VEL
LIN {X 0,Y 545.649,Z 324.679,A -85,B 0,C 180,E1 -3707.746,E2 -3707.746} C_VEL
LIN {X 0,Y 545.975,Z 304.509,A -85,B 0,C 180,E1 -3710.731,E2 -3710.731} C_VEL
LIN {X 0,Y 546.204,Z 288.732,A -85,B 0,C 180,E1 -3713.106,E2 -3713.106} C_VEL
LIN {X 0,Y 545.115,Z 282.587,A -85,B 0,C 180,E1 -3714.12,E2 -3714.12} C_VEL
LIN {X 0,Y 545.093,Z 282.581,A -85,B 0,C 180,E1 -3717.173,E2 -3717.173} C_VEL
LIN {X 0,Y 545.065,Z 282.586,A -85,B 0,C 180,E1 -3719.338,E2 -3719.338} C_VEL
LIN {X 0,Y 545.055,Z 282.591,A -85,B 0,C 180,E1 -3721.914,E2 -3721.914} C_VEL
LIN {X 0,Y 545.062,Z 282.588,A -85,B 0,C 180,E1 -3724.564,E2 -3724.564} C_VEL
LIN {X 0,Y 545.035,Z 282.587,A -85,B 0,C 180,E1 -3727.303,E2 -3727.303} C_VEL
LIN {X 0,Y 545.065,Z 282.59,A -85,B 0,C 180,E1 -3730.142,E2 -3730.142} C_VEL
LIN {X 0,Y 545.077,Z 282.583,A -85,B 0,C 180,E1 -3733.106,E2 -3733.106} C_VEL
LIN {X 0,Y 545.047,Z 282.59,A -85,B 0,C 180,E1 -3736.226,E2 -3736.226} C_VEL
LIN {X 0,Y 545.085,Z 282.586,A -85,B 0,C 180,E1 -3738.885,E2 -3738.885} C_VEL
LIN {X 0,Y 545.049,Z 282.585,A -85,B 0,C 180,E1 -3741.762,E2 -3741.762} C_VEL
LIN {X 0,Y 545.039,Z 282.593,A -85,B 0,C 180,E1 -3744.531,E2 -3744.531} C_VEL
LIN {X 0,Y 545.066,Z 282.587,A -85,B 0,C 180,E1 -3747.211,E2 -3747.211} C_VEL
LIN {X 0,Y 545.063,Z 282.583,A -85,B 0,C 180,E1 -3749.81,E2 -3749.81} C_VEL
LIN {X 0,Y 545.085,Z 282.582,A -85,B 0,C 180,E1 -3752.344,E2 -3752.344} C_VEL
LIN {X 0,Y 545.113,Z 282.584,A -85,B 0,C 180,E1 -3754.82,E2 -3754.82} C_VEL
LIN {X 0,Y 545.04,Z 282.594,A -85,B 0,C 180,E1 -3757.242,E2 -3757.242} C_VEL
LIN {X 0,Y 545.116,Z 282.577,A -85,B 0,C 180,E1 -3760.415,E2 -3760.415} C_VEL
LIN {X 0,Y 545.068,Z 282.589,A -85,B 0,C 180,E1 -3763.521,E2 -3763.521} C_VEL
LIN {X 0,Y 545.09,Z 282.583,A -85,B 0,C 180,E1 -3765.82,E2 -3765.82} C_VEL
LIN {X 0,Y 545.112,Z 282.579,A -85,B 0,C 180,E1 -3768.849,E2 -3768.849} C_VEL
LIN {X 0,Y 545.125,Z 282.58,A -85,B 0,C 180,E1 -3771.847,E2 -3771.847} C_VEL
LIN {X 0,Y 545.2,Z 282.567,A -85,B 0,C 180,E1 -3774.823,E2 -3774.823} C_VEL
LIN {X 0,Y 545.186,Z 282.576,A -85,B 0,C 180,E1 -3777.783,E2 -3777.783} C_VEL
LIN {X 0,Y 545.204,Z 282.566,A -85,B 0,C 180,E1 -3780.738,E2 -3780.738} C_VEL
LIN {X 0,Y 545.165,Z 282.571,A -85,B 0,C 180,E1 -3782.956,E2 -3782.956} C_VEL
LIN {X 0,Y 545.161,Z 282.581,A -85,B 0,C 180,E1 -3785.919,E2 -3785.919} C_VEL
LIN {X 0,Y 545.111,Z 282.577,A -85,B 0,C 180,E1 -3788.9,E2 -3788.9} C_VEL
LIN {X 0,Y 545.129,Z 282.583,A -85,B 0,C 180,E1 -3791.904,E2 -3791.904} C_VEL
LIN {X 0,Y 545.075,Z 282.582,A -85,B 0,C 180,E1 -3794.944,E2 -3794.944} C_VEL
LIN {X 0,Y 545.064,Z 282.59,A -85,B 0,C 180,E1 -3798.026,E2 -3798.026} C_VEL
LIN {X 0,Y 545.086,Z 282.589,A -85,B 0,C 180,E1 -3800.372,E2 -3800.372} C_VEL
LIN {X 0,Y 545.073,Z 282.582,A -85,B 0,C 180,E1 -3803.56,E2 -3803.56} C_VEL
LIN {X 0,Y 545.071,Z 282.586,A -85,B 0,C 180,E1 -3806.001,E2 -3806.001} C_VEL
LIN {X 0,Y 545.082,Z 282.587,A -85,B 0,C 180,E1 -3808.748,E2 -3808.748} C_VEL
LIN {X 0,Y 545.052,Z 282.585,A -85,B 0,C 180,E1 -3811.679,E2 -3811.679} C_VEL
LIN {X 0,Y 545.056,Z 282.593,A -85,B 0,C 180,E1 -3814.565,E2 -3814.565} C_VEL
LIN {X 0,Y 545.057,Z 282.59,A -85,B 0,C 180,E1 -3816.988,E2 -3816.988} C_VEL
LIN {X 0,Y 544.346,Z 282.675,A -85,B 0,C 180,E1 -3817.605,E2 -3817.605} C_VEL
LIN {X 0,Y 541.475,Z 283.038,A -85,B 0,C 180,E1 -3818.606,E2 -3818.606} C_VEL
LIN {X 0,Y 539.085,Z 283.331,A -85,B 0,C 180,E1 -3819.411,E2 -3819.411} C_VEL
LIN {X 0,Y 538.078,Z 283.454,A -85,B 0,C 180,E1 -3820.034,E2 -3820.034} C_VEL
LIN {X 0,Y 538.004,Z 283.464,A -85,B 0,C 180,E1 -3820.244,E2 -3820.244} C_VEL
LIN {X 0,Y 538.022,Z 283.469,A -85,B 0,C 180,E1 -3822.988,E2 -3822.988} C_VEL
LIN {X 0,Y 538.014,Z 283.461,A -85,B 0,C 180,E1 -3825.927,E2 -3825.927} C_VEL
LIN {X 0,Y 537.998,Z 283.471,A -85,B 0,C 180,E1 -3829.22,E2 -3829.22} C_VEL
LIN {X 0,Y 537.985,Z 283.465,A -85,B 0,C 180,E1 -3832.122,E2 -3832.122} C_VEL
LIN {X 0,Y 537.993,Z 283.469,A -85,B 0,C 180,E1 -3834.916,E2 -3834.916} C_VEL
LIN {X 0,Y 538.012,Z 283.466,A -85,B 0,C 180,E1 -3837.617,E2 -3837.617} C_VEL
LIN {X 0,Y 538.001,Z 283.463,A -85,B 0,C 180,E1 -3840.238,E2 -3840.238} C_VEL
LIN {X 0,Y 538.001,Z 283.464,A -85,B 0,C 180,E1 -3842.793,E2 -3842.793} C_VEL
LIN {X 0,Y 537.981,Z 283.472,A -85,B 0,C 180,E1 -3845.29,E2 -3845.29} C_VEL
LIN {X 0,Y 538.013,Z 283.465,A -85,B 0,C 180,E1 -3848.043,E2 -3848.043} C_VEL
LIN {X 0,Y 538.079,Z 283.456,A -85,B 0,C 180,E1 -3850.148,E2 -3850.148} C_VEL
LIN {X 0,Y 537.986,Z 283.468,A -85,B 0,C 180,E1 -3853.298,E2 -3853.298} C_VEL
LIN {X 0,Y 538.058,Z 283.463,A -85,B 0,C 180,E1 -3855.631,E2 -3855.631} C_VEL
LIN {X 0,Y 538.022,Z 283.464,A -85,B 0,C 180,E1 -3858.701,E2 -3858.701} C_VEL
LIN {X 0,Y 538.038,Z 283.53,A -85,B 0,C 180,E1 -3860.603,E2 -3860.603} C_VEL
LIN {X 0,Y 538.388,Z 289.627,A -85,B 0,C 180,E1 -3861.745,E2 -3861.745} C_VEL
LIN {X 0,Y 538.22,Z 304.85,A -85,B 0,C 180,E1 -3864.568,E2 -3864.568} C_VEL
LIN {X 0,Y 538.169,Z 308.776,A -85,B 0,C 180,E1 -3865.295,E2 -3865.295} C_VEL
LIN {X 0,Y 539.676,Z 317.939,A -85,B 0,C 180,E1 -3865.472,E2 -3865.472} C_VEL
LIN {X 0,Y 539.286,Z 415.947,A -85,B 0,C 180,E1 -3866.802,E2 -3866.802} C_VEL
LIN {X 0,Y 539.146,Z 428.844,A -85,B 0,C 180,E1 -3867.128,E2 -3867.128} C_VEL
LIN {X 0,Y 538.963,Z 441.857,A -85,B 0,C 180,E1 -3867.618,E2 -3867.618} C_VEL
LIN {X 0,Y 538.769,Z 453.613,A -85,B 0,C 180,E1 -3868.225,E2 -3868.225} C_VEL
LIN {X 0,Y 538.424,Z 464.926,A -85,B 0,C 180,E1 -3868.972,E2 -3868.972} C_VEL
LIN {X 0,Y 538.221,Z 475.109,A -85,B 0,C 180,E1 -3869.813,E2 -3869.813} C_VEL
LIN {X 0,Y 538.035,Z 484.303,A -85,B 0,C 180,E1 -3870.749,E2 -3870.749} C_VEL
LIN {X 0,Y 537.846,Z 493.217,A -85,B 0,C 180,E1 -3871.872,E2 -3871.872} C_VEL
LIN {X 0,Y 537.692,Z 500.426,A -85,B 0,C 180,E1 -3872.997,E2 -3872.997} C_VEL
LIN {X 0,Y 537.644,Z 506.212,A -85,B 0,C 180,E1 -3874.123,E2 -3874.123} C_VEL
LIN {X 0,Y 537.576,Z 510.79,A -85,B 0,C 180,E1 -3875.251,E2 -3875.251} C_VEL
LIN {X 0,Y 537.591,Z 514.616,A -85,B 0,C 180,E1 -3876.508,E2 -3876.508} C_VEL
LIN {X 0,Y 537.514,Z 516.784,A -85,B 0,C 180,E1 -3877.513,E2 -3877.513} C_VEL
LIN {X 0,Y 537.504,Z 517.944,A -85,B 0,C 180,E1 -3878.27,E2 -3878.27} C_VEL
LIN {X 0,Y 537.478,Z 519.001,A -85,B 0,C 180,E1 -3879.787,E2 -3879.787} C_VEL
LIN {X 0,Y 537.488,Z 518.949,A -85,B 0,C 180,E1 -3880.548,E2 -3880.548} C_VEL
LIN {X 0,Y 537.538,Z 518.483,A -85,B 0,C 180,E1 -3881.31,E2 -3881.31} C_VEL
LIN {X 0,Y 537.471,Z 517.579,A -85,B 0,C 180,E1 -3882.077,E2 -3882.077} C_VEL
LIN {X 0,Y 537.485,Z 516.271,A -85,B 0,C 180,E1 -3882.844,E2 -3882.844} C_VEL
LIN {X 0,Y 537.551,Z 513.474,A -85,B 0,C 180,E1 -3883.997,E2 -3883.997} C_VEL
LIN {X 0,Y 537.616,Z 509.599,A -85,B 0,C 180,E1 -3885.156,E2 -3885.156} C_VEL
LIN {X 0,Y 537.654,Z 504.521,A -85,B 0,C 180,E1 -3886.322,E2 -3886.322} C_VEL
LIN {X 0,Y 537.79,Z 498.067,A -85,B 0,C 180,E1 -3887.492,E2 -3887.492} C_VEL
LIN {X 0,Y 537.945,Z 489.872,A -85,B 0,C 180,E1 -3888.668,E2 -3888.668} C_VEL
LIN {X 0,Y 538.095,Z 481.427,A -85,B 0,C 180,E1 -3889.653,E2 -3889.653} C_VEL
LIN {X 0,Y 538.358,Z 471.008,A -85,B 0,C 180,E1 -3890.639,E2 -3890.639} C_VEL
LIN {X 0,Y 538.542,Z 460.508,A -85,B 0,C 180,E1 -3891.432,E2 -3891.432} C_VEL
LIN {X 0,Y 538.88,Z 448.572,A -85,B 0,C 180,E1 -3892.145,E2 -3892.145} C_VEL
LIN {X 0,Y 538.965,Z 437.119,A -85,B 0,C 180,E1 -3892.674,E2 -3892.674} C_VEL
LIN {X 0,Y 539.127,Z 424.276,A -85,B 0,C 180,E1 -3893.098,E2 -3893.098} C_VEL
LIN {X 0,Y 539.259,Z 411.14,A -85,B 0,C 180,E1 -3893.371,E2 -3893.371} C_VEL
LIN {X 0,Y 539.613,Z 317.097,A -85,B 0,C 180,E1 -3894.631,E2 -3894.631} C_VEL
LIN {X 0,Y 538.137,Z 308.602,A -85,B 0,C 180,E1 -3894.806,E2 -3894.806} C_VEL
LIN {X 0,Y 538.273,Z 297.864,A -85,B 0,C 180,E1 -3896.773,E2 -3896.773} C_VEL
LIN {X 0,Y 538.385,Z 285.589,A -85,B 0,C 180,E1 -3899.002,E2 -3899.002} C_VEL
LIN {X 0,Y 538.079,Z 283.463,A -85,B 0,C 180,E1 -3899.398,E2 -3899.398} C_VEL
LIN {X 0,Y 538.017,Z 283.471,A -85,B 0,C 180,E1 -3902.383,E2 -3902.383} C_VEL
LIN {X 0,Y 537.998,Z 283.466,A -85,B 0,C 180,E1 -3905.084,E2 -3905.084} C_VEL
LIN {X 0,Y 537.991,Z 283.465,A -85,B 0,C 180,E1 -3907.878,E2 -3907.878} C_VEL
LIN {X 0,Y 538.047,Z 283.464,A -85,B 0,C 180,E1 -3910.776,E2 -3910.776} C_VEL
LIN {X 0,Y 538.002,Z 283.464,A -85,B 0,C 180,E1 -3913.816,E2 -3913.816} C_VEL
LIN {X 0,Y 538.025,Z 283.466,A -85,B 0,C 180,E1 -3917.013,E2 -3917.013} C_VEL
LIN {X 0,Y 538.047,Z 283.46,A -85,B 0,C 180,E1 -3919.253,E2 -3919.253} C_VEL
LIN {X 0,Y 537.991,Z 283.464,A -85,B 0,C 180,E1 -3922.122,E2 -3922.122} C_VEL
LIN {X 0,Y 538.001,Z 283.472,A -85,B 0,C 180,E1 -3924.916,E2 -3924.916} C_VEL
LIN {X 0,Y 538.017,Z 283.461,A -85,B 0,C 180,E1 -3927.617,E2 -3927.617} C_VEL
LIN {X 0,Y 538.016,Z 283.46,A -85,B 0,C 180,E1 -3930.239,E2 -3930.239} C_VEL
LIN {X 0,Y 538.056,Z 283.458,A -85,B 0,C 180,E1 -3932.796,E2 -3932.796} C_VEL
LIN {X 0,Y 538.047,Z 283.465,A -85,B 0,C 180,E1 -3935.293,E2 -3935.293} C_VEL
LIN {X 0,Y 538.021,Z 283.46,A -85,B 0,C 180,E1 -3938.546,E2 -3938.546} C_VEL
LIN {X 0,Y 538.032,Z 283.46,A -85,B 0,C 180,E1 -3940.94,E2 -3940.94} C_VEL
LIN {X 0,Y 538.024,Z 283.467,A -85,B 0,C 180,E1 -3943.299,E2 -3943.299} C_VEL
LIN {X 0,Y 538.063,Z 283.465,A -85,B 0,C 180,E1 -3945.631,E2 -3945.631} C_VEL
LIN {X 0,Y 538.076,Z 283.453,A -85,B 0,C 180,E1 -3948.702,E2 -3948.702} C_VEL
LIN {X 0,Y 538.084,Z 283.463,A -85,B 0,C 180,E1 -3951.74,E2 -3951.74} C_VEL
LIN {X 0,Y 538.158,Z 283.443,A -85,B 0,C 180,E1 -3954.755,E2 -3954.755} C_VEL
LIN {X 0,Y 538.167,Z 283.448,A -85,B 0,C 180,E1 -3957.755,E2 -3957.755} C_VEL
LIN {X 0,Y 538.181,Z 283.441,A -85,B 0,C 180,E1 -3960.748,E2 -3960.748} C_VEL
LIN {X 0,Y 538.137,Z 283.444,A -85,B 0,C 180,E1 -3962.995,E2 -3962.995} C_VEL
LIN {X 0,Y 538.119,Z 283.455,A -85,B 0,C 180,E1 -3965.998,E2 -3965.998} C_VEL
LIN {X 0,Y 538.067,Z 283.455,A -85,B 0,C 180,E1 -3969.018,E2 -3969.018} C_VEL
LIN {X 0,Y 538.083,Z 283.455,A -85,B 0,C 180,E1 -3972.063,E2 -3972.063} C_VEL
LIN {X 0,Y 538.045,Z 283.457,A -85,B 0,C 180,E1 -3975.144,E2 -3975.144} C_VEL
LIN {X 0,Y 538.029,Z 283.464,A -85,B 0,C 180,E1 -3978.27,E2 -3978.27} C_VEL
LIN {X 0,Y 538.037,Z 283.466,A -85,B 0,C 180,E1 -3980.652,E2 -3980.652} C_VEL
LIN {X 0,Y 538.004,Z 283.462,A -85,B 0,C 180,E1 -3983.889,E2 -3983.889} C_VEL
LIN {X 0,Y 538.042,Z 283.461,A -85,B 0,C 180,E1 -3986.367,E2 -3986.367} C_VEL
LIN {X 0,Y 538.031,Z 283.468,A -85,B 0,C 180,E1 -3988.934,E2 -3988.934} C_VEL
LIN {X 0,Y 538.01,Z 283.461,A -85,B 0,C 180,E1 -3991.887,E2 -3991.887} C_VEL
LIN {X 0,Y 538.012,Z 283.465,A -85,B 0,C 180,E1 -3994.618,E2 -3994.618} C_VEL
LIN {X 0,Y 538.005,Z 283.472,A -85,B 0,C 180,E1 -3997.17,E2 -3997.17} C_VEL
LIN {X 0,Y 538.023,Z 283.458,A -85,B 0,C 180,E1 -3999.797,E2 -3999.797} C_VEL
LIN {X 0,Y 538.02,Z 283.463,A -85,B 0,C 180,E1 -4002.786,E2 -4002.786} C_VEL
LIN {X 0,Y 538.019,Z 283.464,A -85,B 0,C 180,E1 -4005.927,E2 -4005.927} C_VEL
LIN {X 0,Y 538.032,Z 283.461,A -85,B 0,C 180,E1 -4008.227,E2 -4008.227} C_VEL
LIN {X 0,Y 538.014,Z 283.465,A -85,B 0,C 180,E1 -4011.17,E2 -4011.17} C_VEL
LIN {X 0,Y 537.996,Z 283.469,A -85,B 0,C 180,E1 -4014.089,E2 -4014.089} C_VEL
LIN {X 0,Y 538.033,Z 283.461,A -85,B 0,C 180,E1 -4016.728,E2 -4016.728} C_VEL
LIN {X 0,Y 538.029,Z 283.466,A -85,B 0,C 180,E1 -4019.556,E2 -4019.556} C_VEL
LIN {X 0,Y 538.039,Z 283.467,A -85,B 0,C 180,E1 -4021.95,E2 -4021.95} C_VEL
LIN {X 0,Y 538.066,Z 283.462,A -85,B 0,C 180,E1 -4024.467,E2 -4024.467} C_VEL
LIN {X 0,Y 538.1,Z 283.625,A -85,B 0,C 180,E1 -4025.819,E2 -4025.819} C_VEL
LIN {X 0,Y 539.296,Z 290.898,A -85,B 0,C 180,E1 -4026.986,E2 -4026.986} C_VEL
LIN {X 0,Y 538.927,Z 310.74,A -85,B 0,C 180,E1 -4029.986,E2 -4029.986} C_VEL
LIN {X 0,Y 538.583,Z 329.145,A -85,B 0,C 180,E1 -4032.73,E2 -4032.73} C_VEL
LIN {X 0,Y 538.328,Z 346.127,A -85,B 0,C 180,E1 -4035.238,E2 -4035.238} C_VEL
LIN {X 0,Y 539.636,Z 355.014,A -85,B 0,C 180,E1 -4035.401,E2 -4035.401} C_VEL
LIN {X 0,Y 539.291,Z 454.504,A -85,B 0,C 180,E1 -4036.745,E2 -4036.745} C_VEL
LIN {X 0,Y 539.155,Z 467.813,A -85,B 0,C 180,E1 -4037.077,E2 -4037.077} C_VEL
LIN {X 0,Y 538.94,Z 480.003,A -85,B 0,C 180,E1 -4037.527,E2 -4037.527} C_VEL
LIN {X 0,Y 538.768,Z 491.451,A -85,B 0,C 180,E1 -4038.094,E2 -4038.094} C_VEL
LIN {X 0,Y 538.549,Z 502.629,A -85,B 0,C 180,E1 -4038.807,E2 -4038.807} C_VEL
LIN {X 0,Y 538.254,Z 513.314,A -85,B 0,C 180,E1 -4039.657,E2 -4039.657} C_VEL
LIN {X 0,Y 538.067,Z 522.946,A -85,B 0,C 180,E1 -4040.603,E2 -4040.603} C_VEL
LIN {X 0,Y 537.913,Z 530.842,A -85,B 0,C 180,E1 -4041.548,E2 -4041.548} C_VEL
LIN {X 0,Y 537.755,Z 538.554,A -85,B 0,C 180,E1 -4042.679,E2 -4042.679} C_VEL
LIN {X 0,Y 537.696,Z 545.666,A -85,B 0,C 180,E1 -4043.998,E2 -4043.998} C_VEL
LIN {X 0,Y 537.54,Z 550.372,A -85,B 0,C 180,E1 -4045.125,E2 -4045.125} C_VEL
LIN {X 0,Y 537.591,Z 553.957,A -85,B 0,C 180,E1 -4046.252,E2 -4046.252} C_VEL
LIN {X 0,Y 537.551,Z 555.806,A -85,B 0,C 180,E1 -4047.002,E2 -4047.002} C_VEL
LIN {X 0,Y 537.451,Z 558.181,A -85,B 0,C 180,E1 -4048.501,E2 -4048.501} C_VEL
LIN {X 0,Y 537.442,Z 559,A -85,B 0,C 180,E1 -4050,E2 -4050} C_VEL
LIN {X 0,Y 537.451,Z 558.183,A -85,B 0,C 180,E1 -4051.498,E2 -4051.498} C_VEL
LIN {X 0,Y 537.551,Z 555.811,A -85,B 0,C 180,E1 -4052.997,E2 -4052.997} C_VEL
LIN {X 0,Y 537.603,Z 552.896,A -85,B 0,C 180,E1 -4054.123,E2 -4054.123} C_VEL
LIN {X 0,Y 537.587,Z 548.948,A -85,B 0,C 180,E1 -4055.25,E2 -4055.25} C_VEL
LIN {X 0,Y 537.643,Z 544.102,A -85,B 0,C 180,E1 -4056.326,E2 -4056.326} C_VEL
LIN {X 0,Y 537.772,Z 537.396,A -85,B 0,C 180,E1 -4057.509,E2 -4057.509} C_VEL
LIN {X 0,Y 537.942,Z 529.356,A -85,B 0,C 180,E1 -4058.641,E2 -4058.641} C_VEL
LIN {X 0,Y 538.115,Z 521.165,A -85,B 0,C 180,E1 -4059.585,E2 -4059.585} C_VEL
LIN {X 0,Y 538.345,Z 511.178,A -85,B 0,C 180,E1 -4060.531,E2 -4060.531} C_VEL
LIN {X 0,Y 538.597,Z 501.33,A -85,B 0,C 180,E1 -4061.287,E2 -4061.287} C_VEL
LIN {X 0,Y 538.737,Z 490.127,A -85,B 0,C 180,E1 -4061.979,E2 -4061.979} C_VEL
LIN {X 0,Y 538.958,Z 477.753,A -85,B 0,C 180,E1 -4062.568,E2 -4062.568} C_VEL
LIN {X 0,Y 539.147,Z 464.703,A -85,B 0,C 180,E1 -4063.018,E2 -4063.018} C_VEL
LIN {X 0,Y 539.339,Z 451.693,A -85,B 0,C 180,E1 -4063.301,E2 -4063.301} C_VEL
LIN {X 0,Y 539.602,Z 355.075,A -85,B 0,C 180,E1 -4064.599,E2 -4064.599} C_VEL
LIN {X 0,Y 538.343,Z 346.073,A -85,B 0,C 180,E1 -4064.775,E2 -4064.775} C_VEL
LIN {X 0,Y 538.697,Z 323.735,A -85,B 0,C 180,E1 -4068.086,E2 -4068.086} C_VEL
LIN {X 0,Y 539.009,Z 305.577,A -85,B 0,C 180,E1 -4070.812,E2 -4070.812} C_VEL
LIN {X 0,Y 539.329,Z 291.12,A -85,B 0,C 180,E1 -4073.012,E2 -4073.012} C_VEL
LIN {X 0,Y 538.062,Z 283.465,A -85,B 0,C 180,E1 -4074.266,E2 -4074.266} C_VEL
LIN {X 0,Y 538.058,Z 283.458,A -85,B 0,C 180,E1 -4077.351,E2 -4077.351} C_VEL
LIN {X 0,Y 538.017,Z 283.468,A -85,B 0,C 180,E1 -4079.761,E2 -4079.761} C_VEL
LIN {X 0,Y 538.018,Z 283.467,A -85,B 0,C 180,E1 -4082.382,E2 -4082.382} C_VEL
LIN {X 0,Y 537.998,Z 283.464,A -85,B 0,C 180,E1 -4085.084,E2 -4085.084} C_VEL
LIN {X 0,Y 537.991,Z 283.468,A -85,B 0,C 180,E1 -4087.877,E2 -4087.877} C_VEL
LIN {X 0,Y 538.048,Z 283.461,A -85,B 0,C 180,E1 -4090.775,E2 -4090.775} C_VEL
LIN {X 0,Y 538.002,Z 283.464,A -85,B 0,C 180,E1 -4093.815,E2 -4093.815} C_VEL
LIN {X 0,Y 538.024,Z 283.463,A -85,B 0,C 180,E1 -4097.012,E2 -4097.012} C_VEL
LIN {X 0,Y 538.046,Z 283.459,A -85,B 0,C 180,E1 -4099.252,E2 -4099.252} C_VEL
LIN {X 0,Y 537.989,Z 283.466,A -85,B 0,C 180,E1 -4102.122,E2 -4102.122} C_VEL
LIN {X 0,Y 537.999,Z 283.471,A -85,B 0,C 180,E1 -4104.915,E2 -4104.915} C_VEL
LIN {X 0,Y 538.016,Z 283.462,A -85,B 0,C 180,E1 -4107.617,E2 -4107.617} C_VEL
LIN {X 0,Y 538.015,Z 283.462,A -85,B 0,C 180,E1 -4110.238,E2 -4110.238} C_VEL
LIN {X 0,Y 538.059,Z 283.463,A -85,B 0,C 180,E1 -4112.796,E2 -4112.796} C_VEL
LIN {X 0,Y 538.045,Z 283.464,A -85,B 0,C 180,E1 -4115.292,E2 -4115.292} C_VEL
LIN {X 0,Y 538.011,Z 283.462,A -85,B 0,C 180,E1 -4118.041,E2 -4118.041} C_VEL
LIN {X 0,Y 538.033,Z 283.465,A -85,B 0,C 180,E1 -4120.94,E2 -4120.94} C_VEL
LIN {X 0,Y 538.02,Z 283.471,A -85,B 0,C 180,E1 -4123.299,E2 -4123.299} C_VEL
LIN {X 0,Y 538.059,Z 283.461,A -85,B 0,C 180,E1 -4125.63,E2 -4125.63} C_VEL
LIN {X 0,Y 538.072,Z 283.455,A -85,B 0,C 180,E1 -4128.701,E2 -4128.701} C_VEL
LIN {X 0,Y 538.082,Z 283.459,A -85,B 0,C 180,E1 -4131.739,E2 -4131.739} C_VEL
LIN {X 0,Y 538.157,Z 283.444,A -85,B 0,C 180,E1 -4134.755,E2 -4134.755} C_VEL
LIN {X 0,Y 538.159,Z 283.452,A -85,B 0,C 180,E1 -4137.755,E2 -4137.755} C_VEL
LIN {X 0,Y 538.175,Z 283.441,A -85,B 0,C 180,E1 -4140.748,E2 -4140.748} C_VEL
LIN {X 0,Y 538.132,Z 283.447,A -85,B 0,C 180,E1 -4142.994,E2 -4142.994} C_VEL
LIN {X 0,Y 538.111,Z 283.458,A -85,B 0,C 180,E1 -4145.997,E2 -4145.997} C_VEL
LIN {X 0,Y 538.062,Z 283.455,A -85,B 0,C 180,E1 -4149.018,E2 -4149.018} C_VEL
LIN {X 0,Y 538.077,Z 283.464,A -85,B 0,C 180,E1 -4152.063,E2 -4152.063} C_VEL
LIN {X 0,Y 538.037,Z 283.458,A -85,B 0,C 180,E1 -4155.144,E2 -4155.144} C_VEL
LIN {X 0,Y 538.019,Z 283.471,A -85,B 0,C 180,E1 -4158.27,E2 -4158.27} C_VEL
LIN {X 0,Y 538.031,Z 283.464,A -85,B 0,C 180,E1 -4160.652,E2 -4160.652} C_VEL
LIN {X 0,Y 537.996,Z 283.466,A -85,B 0,C 180,E1 -4163.889,E2 -4163.889} C_VEL
LIN {X 0,Y 538.031,Z 283.468,A -85,B 0,C 180,E1 -4166.367,E2 -4166.367} C_VEL
LIN {X 0,Y 538.024,Z 283.464,A -85,B 0,C 180,E1 -4168.933,E2 -4168.933} C_VEL
LIN {X 0,Y 538.004,Z 283.463,A -85,B 0,C 180,E1 -4171.887,E2 -4171.887} C_VEL
LIN {X 0,Y 538.006,Z 283.472,A -85,B 0,C 180,E1 -4174.618,E2 -4174.618} C_VEL
LIN {X 0,Y 537.998,Z 283.467,A -85,B 0,C 180,E1 -4177.17,E2 -4177.17} C_VEL
LIN {X 0,Y 538.004,Z 283.464,A -85,B 0,C 180,E1 -4180.244,E2 -4180.244} C_VEL
LIN {X 0,Y 537.36,Z 283.553,A -85,B 0,C 180,E1 -4180.869,E2 -4180.869} C_VEL
LIN {X 0,Y 534.51,Z 283.907,A -85,B 0,C 180,E1 -4181.884,E2 -4181.884} C_VEL
LIN {X 0,Y 532.084,Z 284.207,A -85,B 0,C 180,E1 -4182.702,E2 -4182.702} C_VEL
LIN {X 0,Y 531.036,Z 284.335,A -85,B 0,C 180,E1 -4183.333,E2 -4183.333} C_VEL
LIN {X 0,Y 530.948,Z 284.343,A -85,B 0,C 180,E1 -4183.546,E2 -4183.546} C_VEL
LIN {X 0,Y 530.94,Z 284.345,A -85,B 0,C 180,E1 -4186.504,E2 -4186.504} C_VEL
LIN {X 0,Y 530.946,Z 284.345,A -85,B 0,C 180,E1 -4189.565,E2 -4189.565} C_VEL
LIN {X 0,Y 530.963,Z 284.342,A -85,B 0,C 180,E1 -4192.578,E2 -4192.578} C_VEL
LIN {X 0,Y 530.976,Z 284.347,A -85,B 0,C 180,E1 -4195.31,E2 -4195.31} C_VEL
LIN {X 0,Y 530.962,Z 284.341,A -85,B 0,C 180,E1 -4198.032,E2 -4198.032} C_VEL
LIN {X 0,Y 530.984,Z 284.34,A -85,B 0,C 180,E1 -4200.875,E2 -4200.875} C_VEL
LIN {X 0,Y 530.959,Z 284.342,A -85,B 0,C 180,E1 -4204.101,E2 -4204.101} C_VEL
LIN {X 0,Y 530.948,Z 284.342,A -85,B 0,C 180,E1 -4206.603,E2 -4206.603} C_VEL
LIN {X 0,Y 530.996,Z 284.338,A -85,B 0,C 180,E1 -4209.062,E2 -4209.062} C_VEL
LIN {X 0,Y 530.97,Z 284.346,A -85,B 0,C 180,E1 -4211.479,E2 -4211.479} C_VEL
LIN {X 0,Y 530.989,Z 284.337,A -85,B 0,C 180,E1 -4214.65,E2 -4214.65} C_VEL
LIN {X 0,Y 531.012,Z 284.344,A -85,B 0,C 180,E1 -4217.775,E2 -4217.775} C_VEL
LIN {X 0,Y 531.017,Z 284.514,A -85,B 0,C 180,E1 -4220.526,E2 -4220.526} C_VEL
LIN {X 0,Y 531.449,Z 289.348,A -85,B 0,C 180,E1 -4221.445,E2 -4221.445} C_VEL
LIN {X 0,Y 531.211,Z 305.735,A -85,B 0,C 180,E1 -4224.496,E2 -4224.496} C_VEL
LIN {X 0,Y 531.245,Z 308.901,A -85,B 0,C 180,E1 -4225.091,E2 -4225.091} C_VEL
LIN {X 0,Y 532.83,Z 319.258,A -85,B 0,C 180,E1 -4225.295,E2 -4225.295} C_VEL
LIN {X 0,Y 532.398,Z 415.762,A -85,B 0,C 180,E1 -4226.618,E2 -4226.618} C_VEL
LIN {X 0,Y 532.237,Z 428.813,A -85,B 0,C 180,E1 -4226.949,E2 -4226.949} C_VEL
LIN {X 0,Y 532.058,Z 441.897,A -85,B 0,C 180,E1 -4227.445,E2 -4227.445} C_VEL
LIN {X 0,Y 531.822,Z 452.952,A -85,B 0,C 180,E1 -4228.012,E2 -4228.012} C_VEL
LIN {X 0,Y 531.481,Z 464.428,A -85,B 0,C 180,E1 -4228.769,E2 -4228.769} C_VEL
LIN {X 0,Y 531.226,Z 474.748,A -85,B 0,C 180,E1 -4229.621,E2 -4229.621} C_VEL
LIN {X 0,Y 531.042,Z 484.072,A -85,B 0,C 180,E1 -4230.569,E2 -4230.569} C_VEL
LIN {X 0,Y 530.823,Z 493.081,A -85,B 0,C 180,E1 -4231.707,E2 -4231.707} C_VEL
LIN {X 0,Y 530.679,Z 500.355,A -85,B 0,C 180,E1 -4232.847,E2 -4232.847} C_VEL
LIN {X 0,Y 530.559,Z 507.069,A -85,B 0,C 180,E1 -4234.178,E2 -4234.178} C_VEL
LIN {X 0,Y 530.507,Z 511.509,A -85,B 0,C 180,E1 -4235.321,E2 -4235.321} C_VEL
LIN {X 0,Y 530.524,Z 515.002,A -85,B 0,C 180,E1 -4236.514,E2 -4236.514} C_VEL
LIN {X 0,Y 530.424,Z 517.293,A -85,B 0,C 180,E1 -4237.614,E2 -4237.614} C_VEL
LIN {X 0,Y 530.414,Z 518.349,A -85,B 0,C 180,E1 -4238.381,E2 -4238.381} C_VEL
LIN {X 0,Y 530.387,Z 519.293,A -85,B 0,C 180,E1 -4239.919,E2 -4239.919} C_VEL
LIN {X 0,Y 530.446,Z 518.722,A -85,B 0,C 180,E1 -4241.351,E2 -4241.351} C_VEL
LIN {X 0,Y 530.384,Z 517.643,A -85,B 0,C 180,E1 -4242.24,E2 -4242.24} C_VEL
LIN {X 0,Y 530.396,Z 516.276,A -85,B 0,C 180,E1 -4243.018,E2 -4243.018} C_VEL
LIN {X 0,Y 530.476,Z 513.357,A -85,B 0,C 180,E1 -4244.188,E2 -4244.188} C_VEL
LIN {X 0,Y 530.547,Z 509.351,A -85,B 0,C 180,E1 -4245.363,E2 -4245.363} C_VEL
LIN {X 0,Y 530.642,Z 503.089,A -85,B 0,C 180,E1 -4246.742,E2 -4246.742} C_VEL
LIN {X 0,Y 530.8,Z 496.175,A -85,B 0,C 180,E1 -4247.929,E2 -4247.929} C_VEL
LIN {X 0,Y 530.942,Z 489.052,A -85,B 0,C 180,E1 -4248.923,E2 -4248.923} C_VEL
LIN {X 0,Y 531.128,Z 480.184,A -85,B 0,C 180,E1 -4249.943,E2 -4249.943} C_VEL
LIN {X 0,Y 531.39,Z 469.542,A -85,B 0,C 180,E1 -4250.922,E2 -4250.922} C_VEL
LIN {X 0,Y 531.658,Z 458.679,A -85,B 0,C 180,E1 -4251.724,E2 -4251.724} C_VEL
LIN {X 0,Y 531.953,Z 447.833,A -85,B 0,C 180,E1 -4252.359,E2 -4252.359} C_VEL
LIN {X 0,Y 532.107,Z 436.33,A -85,B 0,C 180,E1 -4252.88,E2 -4252.88} C_VEL
LIN {X 0,Y 532.283,Z 422.991,A -85,B 0,C 180,E1 -4253.309,E2 -4253.309} C_VEL
LIN {X 0,Y 532.374,Z 410.386,A -85,B 0,C 180,E1 -4253.563,E2 -4253.563} C_VEL
LIN {X 0,Y 532.796,Z 318.153,A -85,B 0,C 180,E1 -4254.811,E2 -4254.811} C_VEL
LIN {X 0,Y 531.137,Z 308.774,A -85,B 0,C 180,E1 -4255.005,E2 -4255.005} C_VEL
LIN {X 0,Y 531.292,Z 293.68,A -85,B 0,C 180,E1 -4257.772,E2 -4257.772} C_VEL
LIN {X 0,Y 531.281,Z 285.899,A -85,B 0,C 180,E1 -4259.182,E2 -4259.182} C_VEL
LIN {X 0,Y 531.029,Z 284.342,A -85,B 0,C 180,E1 -4259.483,E2 -4259.483} C_VEL
LIN {X 0,Y 530.966,Z 284.344,A -85,B 0,C 180,E1 -4262.867,E2 -4262.867} C_VEL
LIN {X 0,Y 530.954,Z 284.343,A -85,B 0,C 180,E1 -4265.62,E2 -4265.62} C_VEL
LIN {X 0,Y 530.965,Z 284.348,A -85,B 0,C 180,E1 -4268.653,E2 -4268.653} C_VEL
LIN {X 0,Y 530.992,Z 284.337,A -85,B 0,C 180,E1 -4271.436,E2 -4271.436} C_VEL
LIN {X 0,Y 530.972,Z 284.347,A -85,B 0,C 180,E1 -4274.548,E2 -4274.548} C_VEL
LIN {X 0,Y 530.981,Z 284.338,A -85,B 0,C 180,E1 -4277.834,E2 -4277.834} C_VEL
LIN {X 0,Y 530.985,Z 284.343,A -85,B 0,C 180,E1 -4280.557,E2 -4280.557} C_VEL
LIN {X 0,Y 530.954,Z 284.342,A -85,B 0,C 180,E1 -4283.442,E2 -4283.442} C_VEL
LIN {X 0,Y 530.998,Z 284.337,A -85,B 0,C 180,E1 -4286.494,E2 -4286.494} C_VEL
LIN {X 0,Y 530.973,Z 284.343,A -85,B 0,C 180,E1 -4289.355,E2 -4289.355} C_VEL
LIN {X 0,Y 531.011,Z 284.332,A -85,B 0,C 180,E1 -4292.468,E2 -4292.468} C_VEL
LIN {X 0,Y 531.004,Z 284.338,A -85,B 0,C 180,E1 -4294.943,E2 -4294.943} C_VEL
LIN {X 0,Y 530.97,Z 284.339,A -85,B 0,C 180,E1 -4298.247,E2 -4298.247} C_VEL
LIN {X 0,Y 530.991,Z 284.335,A -85,B 0,C 180,E1 -4300.677,E2 -4300.677} C_VEL
LIN {X 0,Y 530.985,Z 284.341,A -85,B 0,C 180,E1 -4303.071,E2 -4303.071} C_VEL
LIN {X 0,Y 531.018,Z 284.339,A -85,B 0,C 180,E1 -4305.436,E2 -4305.436} C_VEL
LIN {X 0,Y 531.035,Z 284.33,A -85,B 0,C 180,E1 -4308.55,E2 -4308.55} C_VEL
LIN {X 0,Y 531.054,Z 284.336,A -85,B 0,C 180,E1 -4311.63,E2 -4311.63} C_VEL
LIN {X 0,Y 531.117,Z 284.321,A -85,B 0,C 180,E1 -4314.685,E2 -4314.685} C_VEL
LIN {X 0,Y 531.139,Z 284.323,A -85,B 0,C 180,E1 -4317.725,E2 -4317.725} C_VEL
LIN {X 0,Y 531.151,Z 284.317,A -85,B 0,C 180,E1 -4320.758,E2 -4320.758} C_VEL
LIN {X 0,Y 531.104,Z 284.32,A -85,B 0,C 180,E1 -4323.034,E2 -4323.034} C_VEL
LIN {X 0,Y 531.075,Z 284.333,A -85,B 0,C 180,E1 -4326.077,E2 -4326.077} C_VEL
LIN {X 0,Y 531.054,Z 284.337,A -85,B 0,C 180,E1 -4328.371,E2 -4328.371} C_VEL
LIN {X 0,Y 531.051,Z 284.327,A -85,B 0,C 180,E1 -4331.672,E2 -4331.672} C_VEL
LIN {X 0,Y 531.031,Z 284.333,A -85,B 0,C 180,E1 -4334.956,E2 -4334.956} C_VEL
LIN {X 0,Y 531.017,Z 284.333,A -85,B 0,C 180,E1 -4337.723,E2 -4337.723} C_VEL
LIN {X 0,Y 531.024,Z 284.334,A -85,B 0,C 180,E1 -4340.127,E2 -4340.127} C_VEL
LIN {X 0,Y 530.946,Z 284.349,A -85,B 0,C 180,E1 -4342.574,E2 -4342.574} C_VEL
LIN {X 0,Y 531.006,Z 284.34,A -85,B 0,C 180,E1 -4345.058,E2 -4345.058} C_VEL
LIN {X 0,Y 531.013,Z 284.334,A -85,B 0,C 180,E1 -4347.596,E2 -4347.596} C_VEL
LIN {X 0,Y 530.974,Z 284.343,A -85,B 0,C 180,E1 -4350.645,E2 -4350.645} C_VEL
LIN {X 0,Y 530.987,Z 284.338,A -85,B 0,C 180,E1 -4353.773,E2 -4353.773} C_VEL
LIN {X 0,Y 530.956,Z 284.341,A -85,B 0,C 180,E1 -4356.559,E2 -4356.559} C_VEL
LIN {X 0,Y 530.986,Z 284.339,A -85,B 0,C 180,E1 -4359.444,E2 -4359.444} C_VEL
LIN {X 0,Y 530.979,Z 284.338,A -85,B 0,C 180,E1 -4362.457,E2 -4362.457} C_VEL
LIN {X 0,Y 530.977,Z 284.346,A -85,B 0,C 180,E1 -4365.622,E2 -4365.622} C_VEL
LIN {X 0,Y 530.995,Z 284.336,A -85,B 0,C 180,E1 -4368.565,E2 -4368.565} C_VEL
LIN {X 0,Y 530.958,Z 284.35,A -85,B 0,C 180,E1 -4371.53,E2 -4371.53} C_VEL
LIN {X 0,Y 530.956,Z 284.343,A -85,B 0,C 180,E1 -4374.38,E2 -4374.38} C_VEL
LIN {X 0,Y 530.969,Z 284.342,A -85,B 0,C 180,E1 -4377.134,E2 -4377.134} C_VEL
LIN {X 0,Y 530.972,Z 284.347,A -85,B 0,C 180,E1 -4379.803,E2 -4379.803} C_VEL
LIN {X 0,Y 531.013,Z 284.338,A -85,B 0,C 180,E1 -4382.468,E2 -4382.468} C_VEL
LIN {X 0,Y 531.031,Z 284.339,A -85,B 0,C 180,E1 -4385.57,E2 -4385.57} C_VEL
LIN {X 0,Y 531.061,Z 284.591,A -85,B 0,C 180,E1 -4385.675,E2 -4385.675} C_VEL
LIN {X 0,Y 532.339,Z 291.93,A -85,B 0,C 180,E1 -4386.873,E2 -4386.873} C_VEL
LIN {X 0,Y 531.988,Z 310.457,A -85,B 0,C 180,E1 -4389.714,E2 -4389.714} C_VEL
LIN {X 0,Y 531.567,Z 330.181,A -85,B 0,C 180,E1 -4392.694,E2 -4392.694} C_VEL
LIN {X 0,Y 531.305,Z 345.929,A -85,B 0,C 180,E1 -4395.047,E2 -4395.047} C_VEL
LIN {X 0,Y 532.781,Z 355.917,A -85,B 0,C 180,E1 -4395.225,E2 -4395.225} C_VEL
LIN {X 0,Y 532.39,Z 454.209,A -85,B 0,C 180,E1 -4396.57,E2 -4396.57} C_VEL
LIN {X 0,Y 532.23,Z 467.526,A -85,B 0,C 180,E1 -4396.906,E2 -4396.906} C_VEL
LIN {X 0,Y 531.975,Z 479.719,A -85,B 0,C 180,E1 -4397.361,E2 -4397.361} C_VEL
LIN {X 0,Y 531.768,Z 491.634,A -85,B 0,C 180,E1 -4397.962,E2 -4397.962} C_VEL
LIN {X 0,Y 531.526,Z 503.649,A -85,B 0,C 180,E1 -4398.753,E2 -4398.753} C_VEL
LIN {X 0,Y 531.203,Z 514.112,A -85,B 0,C 180,E1 -4399.615,E2 -4399.615} C_VEL
LIN {X 0,Y 531.019,Z 522.671,A -85,B 0,C 180,E1 -4400.477,E2 -4400.477} C_VEL
LIN {X 0,Y 530.851,Z 530.569,A -85,B 0,C 180,E1 -4401.434,E2 -4401.434} C_VEL
LIN {X 0,Y 530.675,Z 538.283,A -85,B 0,C 180,E1 -4402.581,E2 -4402.581} C_VEL
LIN {X 0,Y 530.588,Z 545.395,A -85,B 0,C 180,E1 -4403.917,E2 -4403.917} C_VEL
LIN {X 0,Y 530.459,Z 550.124,A -85,B 0,C 180,E1 -4405.059,E2 -4405.059} C_VEL
LIN {X 0,Y 530.516,Z 553.743,A -85,B 0,C 180,E1 -4406.202,E2 -4406.202} C_VEL
LIN {X 0,Y 530.457,Z 555.606,A -85,B 0,C 180,E1 -4406.962,E2 -4406.962} C_VEL
LIN {X 0,Y 530.41,Z 557.003,A -85,B 0,C 180,E1 -4407.722,E2 -4407.722} C_VEL
LIN {X 0,Y 530.344,Z 558.608,A -85,B 0,C 180,E1 -4409.24,E2 -4409.24} C_VEL
LIN {X 0,Y 530.345,Z 558.826,A -85,B 0,C 180,E1 -4410,E2 -4410} C_VEL
LIN {X 0,Y 530.361,Z 558.003,A -85,B 0,C 180,E1 -4411.518,E2 -4411.518} C_VEL
LIN {X 0,Y 530.41,Z 557.008,A -85,B 0,C 180,E1 -4412.278,E2 -4412.278} C_VEL
LIN {X 0,Y 530.457,Z 555.613,A -85,B 0,C 180,E1 -4413.038,E2 -4413.038} C_VEL
LIN {X 0,Y 530.522,Z 552.676,A -85,B 0,C 180,E1 -4414.178,E2 -4414.178} C_VEL
LIN {X 0,Y 530.524,Z 548.696,A -85,B 0,C 180,E1 -4415.32,E2 -4415.32} C_VEL
LIN {X 0,Y 530.595,Z 542.987,A -85,B 0,C 180,E1 -4416.578,E2 -4416.578} C_VEL
LIN {X 0,Y 530.73,Z 535.891,A -85,B 0,C 180,E1 -4417.801,E2 -4417.801} C_VEL
LIN {X 0,Y 530.91,Z 527.596,A -85,B 0,C 180,E1 -4418.948,E2 -4418.948} C_VEL
LIN {X 0,Y 531.105,Z 519.094,A -85,B 0,C 180,E1 -4419.905,E2 -4419.905} C_VEL
LIN {X 0,Y 531.358,Z 508.591,A -85,B 0,C 180,E1 -4420.864,E2 -4420.864} C_VEL
LIN {X 0,Y 531.626,Z 497.616,A -85,B 0,C 180,E1 -4421.67,E2 -4421.67} C_VEL
LIN {X 0,Y 531.867,Z 486.815,A -85,B 0,C 180,E1 -4422.302,E2 -4422.302} C_VEL
LIN {X 0,Y 532.064,Z 475.133,A -85,B 0,C 180,E1 -4422.831,E2 -4422.831} C_VEL
LIN {X 0,Y 532.292,Z 461.676,A -85,B 0,C 180,E1 -4423.262,E2 -4423.262} C_VEL
LIN {X 0,Y 532.435,Z 448.375,A -85,B 0,C 180,E1 -4423.525,E2 -4423.525} C_VEL
LIN {X 0,Y 532.744,Z 355.97,A -85,B 0,C 180,E1 -4424.775,E2 -4424.775} C_VEL
LIN {X 0,Y 531.311,Z 345.871,A -85,B 0,C 180,E1 -4424.966,E2 -4424.966} C_VEL
LIN {X 0,Y 531.716,Z 323.659,A -85,B 0,C 180,E1 -4428.304,E2 -4428.304} C_VEL
LIN {X 0,Y 532.125,Z 304.016,A -85,B 0,C 180,E1 -4431.297,E2 -4431.297} C_VEL
LIN {X 0,Y 532.392,Z 292.181,A -85,B 0,C 180,E1 -4433.124,E2 -4433.124} C_VEL
LIN {X 0,Y 531.031,Z 284.339,A -85,B 0,C 180,E1 -4434.43,E2 -4434.43} C_VEL
LIN {X 0,Y 531.016,Z 284.339,A -85,B 0,C 180,E1 -4437.595,E2 -4437.595} C_VEL
LIN {X 0,Y 530.974,Z 284.341,A -85,B 0,C 180,E1 -4440.644,E2 -4440.644} C_VEL
LIN {X 0,Y 530.987,Z 284.34,A -85,B 0,C 180,E1 -4443.772,E2 -4443.772} C_VEL
LIN {X 0,Y 530.954,Z 284.346,A -85,B 0,C 180,E1 -4446.558,E2 -4446.558} C_VEL
LIN {X 0,Y 530.984,Z 284.337,A -85,B 0,C 180,E1 -4449.443,E2 -4449.443} C_VEL
LIN {X 0,Y 530.978,Z 284.348,A -85,B 0,C 180,E1 -4452.456,E2 -4452.456} C_VEL
LIN {X 0,Y 530.975,Z 284.338,A -85,B 0,C 180,E1 -4455.621,E2 -4455.621} C_VEL
LIN {X 0,Y 530.995,Z 284.346,A -85,B 0,C 180,E1 -4458.564,E2 -4458.564} C_VEL
LIN {X 0,Y 530.954,Z 284.341,A -85,B 0,C 180,E1 -4461.529,E2 -4461.529} C_VEL
LIN {X 0,Y 530.953,Z 284.345,A -85,B 0,C 180,E1 -4464.38,E2 -4464.38} C_VEL
LIN {X 0,Y 530.964,Z 284.345,A -85,B 0,C 180,E1 -4467.133,E2 -4467.133} C_VEL
LIN {X 0,Y 530.966,Z 284.339,A -85,B 0,C 180,E1 -4469.803,E2 -4469.803} C_VEL
LIN {X 0,Y 531.011,Z 284.336,A -85,B 0,C 180,E1 -4472.466,E2 -4472.466} C_VEL
LIN {X 0,Y 531.002,Z 284.343,A -85,B 0,C 180,E1 -4474.942,E2 -4474.942} C_VEL
LIN {X 0,Y 530.967,Z 284.339,A -85,B 0,C 180,E1 -4478.246,E2 -4478.246} C_VEL
LIN {X 0,Y 530.991,Z 284.339,A -85,B 0,C 180,E1 -4480.677,E2 -4480.677} C_VEL
LIN {X 0,Y 530.981,Z 284.344,A -85,B 0,C 180,E1 -4483.071,E2 -4483.071} C_VEL
LIN {X 0,Y 531.036,Z 284.339,A -85,B 0,C 180,E1 -4485.436,E2 -4485.436} C_VEL
LIN {X 0,Y 531.031,Z 284.331,A -85,B 0,C 180,E1 -4488.549,E2 -4488.549} C_VEL
LIN {X 0,Y 531.052,Z 284.337,A -85,B 0,C 180,E1 -4491.629,E2 -4491.629} C_VEL
LIN {X 0,Y 531.116,Z 284.321,A -85,B 0,C 180,E1 -4494.685,E2 -4494.685} C_VEL
LIN {X 0,Y 531.131,Z 284.328,A -85,B 0,C 180,E1 -4497.725,E2 -4497.725} C_VEL
LIN {X 0,Y 531.146,Z 284.317,A -85,B 0,C 180,E1 -4500.758,E2 -4500.758} C_VEL
LIN {X 0,Y 531.1,Z 284.323,A -85,B 0,C 180,E1 -4503.034,E2 -4503.034} C_VEL
LIN {X 0,Y 531.065,Z 284.334,A -85,B 0,C 180,E1 -4506.077,E2 -4506.077} C_VEL
LIN {X 0,Y 531.05,Z 284.333,A -85,B 0,C 180,E1 -4508.37,E2 -4508.37} C_VEL
LIN {X 0,Y 531.045,Z 284.334,A -85,B 0,C 180,E1 -4511.672,E2 -4511.672} C_VEL
LIN {X 0,Y 531.023,Z 284.332,A -85,B 0,C 180,E1 -4514.955,E2 -4514.955} C_VEL
LIN {X 0,Y 530.975,Z 284.341,A -85,B 0,C 180,E1 -4517.724,E2 -4517.724} C_VEL
LIN {X 0,Y 531.019,Z 284.341,A -85,B 0,C 180,E1 -4520.127,E2 -4520.127} C_VEL
LIN {X 0,Y 530.939,Z 284.349,A -85,B 0,C 180,E1 -4522.574,E2 -4522.574} C_VEL
LIN {X 0,Y 530.988,Z 284.338,A -85,B 0,C 180,E1 -4525.058,E2 -4525.058} C_VEL
LIN {X 0,Y 530.982,Z 284.337,A -85,B 0,C 180,E1 -4527.597,E2 -4527.597} C_VEL
LIN {X 0,Y 530.968,Z 284.348,A -85,B 0,C 180,E1 -4530.645,E2 -4530.645} C_VEL
LIN {X 0,Y 530.981,Z 284.338,A -85,B 0,C 180,E1 -4533.773,E2 -4533.773} C_VEL
LIN {X 0,Y 530.949,Z 284.349,A -85,B 0,C 180,E1 -4536.559,E2 -4536.559} C_VEL
LIN {X 0,Y 530.965,Z 284.341,A -85,B 0,C 180,E1 -4539.445,E2 -4539.445} C_VEL
LIN {X 0,Y 530.973,Z 284.342,A -85,B 0,C 180,E1 -4542.457,E2 -4542.457} C_VEL
LIN {X 0,Y 530.948,Z 284.343,A -85,B 0,C 180,E1 -4543.546,E2 -4543.546} C_VEL
LIN {X 0,Y 530.278,Z 284.426,A -85,B 0,C 180,E1 -4544.18,E2 -4544.18} C_VEL
LIN {X 0,Y 527.433,Z 284.786,A -85,B 0,C 180,E1 -4545.209,E2 -4545.209} C_VEL
LIN {X 0,Y 525.025,Z 285.09,A -85,B 0,C 180,E1 -4546.037,E2 -4546.037} C_VEL
LIN {X 0,Y 523.982,Z 285.218,A -85,B 0,C 180,E1 -4546.677,E2 -4546.677} C_VEL
LIN {X 0,Y 523.891,Z 285.227,A -85,B 0,C 180,E1 -4546.893,E2 -4546.893} C_VEL
LIN {X 0,Y 523.908,Z 285.219,A -85,B 0,C 180,E1 -4549.918,E2 -4549.918} C_VEL
LIN {X 0,Y 523.903,Z 285.224,A -85,B 0,C 180,E1 -4552.868,E2 -4552.868} C_VEL
LIN {X 0,Y 523.916,Z 285.221,A -85,B 0,C 180,E1 -4555.709,E2 -4555.709} C_VEL
LIN {X 0,Y 523.914,Z 285.218,A -85,B 0,C 180,E1 -4558.456,E2 -4558.456} C_VEL
LIN {X 0,Y 523.921,Z 285.223,A -85,B 0,C 180,E1 -4561.125,E2 -4561.125} C_VEL
LIN {X 0,Y 523.906,Z 285.221,A -85,B 0,C 180,E1 -4563.998,E2 -4563.998} C_VEL
LIN {X 0,Y 523.906,Z 285.22,A -85,B 0,C 180,E1 -4566.27,E2 -4566.27} C_VEL
LIN {X 0,Y 523.943,Z 285.214,A -85,B 0,C 180,E1 -4568.767,E2 -4568.767} C_VEL
LIN {X 0,Y 523.934,Z 285.218,A -85,B 0,C 180,E1 -4571.221,E2 -4571.221} C_VEL
LIN {X 0,Y 523.911,Z 285.227,A -85,B 0,C 180,E1 -4573.639,E2 -4573.639} C_VEL
LIN {X 0,Y 523.928,Z 285.223,A -85,B 0,C 180,E1 -4576.028,E2 -4576.028} C_VEL
LIN {X 0,Y 523.958,Z 285.218,A -85,B 0,C 180,E1 -4578.393,E2 -4578.393} C_VEL
LIN {X 0,Y 523.952,Z 285.272,A -85,B 0,C 180,E1 -4580.397,E2 -4580.397} C_VEL
LIN {X 0,Y 524.456,Z 290.101,A -85,B 0,C 180,E1 -4581.33,E2 -4581.33} C_VEL
LIN {X 0,Y 524.23,Z 305.61,A -85,B 0,C 180,E1 -4584.23,E2 -4584.23} C_VEL
LIN {X 0,Y 524.254,Z 309.287,A -85,B 0,C 180,E1 -4584.905,E2 -4584.905} C_VEL
LIN {X 0,Y 525.923,Z 318.943,A -85,B 0,C 180,E1 -4585.089,E2 -4585.089} C_VEL
LIN {X 0,Y 525.49,Z 416.708,A -85,B 0,C 180,E1 -4586.454,E2 -4586.454} C_VEL
LIN {X 0,Y 525.327,Z 430.267,A -85,B 0,C 180,E1 -4586.813,E2 -4586.813} C_VEL
LIN {X 0,Y 525.111,Z 443.001,A -85,B 0,C 180,E1 -4587.315,E2 -4587.315} C_VEL
LIN {X 0,Y 524.864,Z 455.382,A -85,B 0,C 180,E1 -4587.986,E2 -4587.986} C_VEL
LIN {X 0,Y 524.45,Z 466.477,A -85,B 0,C 180,E1 -4588.753,E2 -4588.753} C_VEL
LIN {X 0,Y 524.205,Z 476.462,A -85,B 0,C 180,E1 -4589.616,E2 -4589.616} C_VEL
LIN {X 0,Y 523.994,Z 485.476,A -85,B 0,C 180,E1 -4590.577,E2 -4590.577} C_VEL
LIN {X 0,Y 523.755,Z 494.284,A -85,B 0,C 180,E1 -4591.73,E2 -4591.73} C_VEL
LIN {X 0,Y 523.611,Z 501.394,A -85,B 0,C 180,E1 -4592.885,E2 -4592.885} C_VEL
LIN {X 0,Y 523.51,Z 506.205,A -85,B 0,C 180,E1 -4593.849,E2 -4593.849} C_VEL
LIN {X 0,Y 523.391,Z 510.899,A -85,B 0,C 180,E1 -4595.007,E2 -4595.007} C_VEL
LIN {X 0,Y 523.41,Z 514.492,A -85,B 0,C 180,E1 -4596.167,E2 -4596.167} C_VEL
LIN {X 0,Y 523.365,Z 516.358,A -85,B 0,C 180,E1 -4596.942,E2 -4596.942} C_VEL
LIN {X 0,Y 523.352,Z 517.757,A -85,B 0,C 180,E1 -4597.718,E2 -4597.718} C_VEL
LIN {X 0,Y 523.319,Z 518.754,A -85,B 0,C 180,E1 -4598.495,E2 -4598.495} C_VEL
LIN {X 0,Y 523.307,Z 519.577,A -85,B 0,C 180,E1 -4600.055,E2 -4600.055} C_VEL
LIN {X 0,Y 523.361,Z 518.958,A -85,B 0,C 180,E1 -4601.396,E2 -4601.396} C_VEL
LIN {X 0,Y 523.29,Z 517.708,A -85,B 0,C 180,E1 -4602.409,E2 -4602.409} C_VEL
LIN {X 0,Y 523.312,Z 516.252,A -85,B 0,C 180,E1 -4603.198,E2 -4603.198} C_VEL
LIN {X 0,Y 523.411,Z 513.215,A -85,B 0,C 180,E1 -4604.383,E2 -4604.383} C_VEL
LIN {X 0,Y 523.492,Z 509.064,A -85,B 0,C 180,E1 -4605.575,E2 -4605.575} C_VEL
LIN {X 0,Y 523.611,Z 502.624,A -85,B 0,C 180,E1 -4606.974,E2 -4606.974} C_VEL
LIN {X 0,Y 523.796,Z 495.542,A -85,B 0,C 180,E1 -4608.177,E2 -4608.177} C_VEL
LIN {X 0,Y 523.932,Z 488.217,A -85,B 0,C 180,E1 -4609.186,E2 -4609.186} C_VEL
LIN {X 0,Y 524.2,Z 478.25,A -85,B 0,C 180,E1 -4610.297,E2 -4610.297} C_VEL
LIN {X 0,Y 524.472,Z 468.083,A -85,B 0,C 180,E1 -4611.211,E2 -4611.211} C_VEL
LIN {X 0,Y 524.755,Z 458.339,A -85,B 0,C 180,E1 -4611.921,E2 -4611.921} C_VEL
LIN {X 0,Y 525.049,Z 447.727,A -85,B 0,C 180,E1 -4612.543,E2 -4612.543} C_VEL
LIN {X 0,Y 525.174,Z 435.451,A -85,B 0,C 180,E1 -4613.096,E2 -4613.096} C_VEL
LIN {X 0,Y 525.35,Z 422.601,A -85,B 0,C 180,E1 -4613.505,E2 -4613.505} C_VEL
LIN {X 0,Y 525.474,Z 409.504,A -85,B 0,C 180,E1 -4613.76,E2 -4613.76} C_VEL
LIN {X 0,Y 525.952,Z 318.874,A -85,B 0,C 180,E1 -4615.001,E2 -4615.001} C_VEL
LIN {X 0,Y 524.181,Z 309.029,A -85,B 0,C 180,E1 -4615.21,E2 -4615.21} C_VEL
LIN {X 0,Y 524.369,Z 292.731,A -85,B 0,C 180,E1 -4618.193,E2 -4618.193} C_VEL
LIN {X 0,Y 524.176,Z 286.29,A -85,B 0,C 180,E1 -4619.367,E2 -4619.367} C_VEL
LIN {X 0,Y 524.005,Z 285.218,A -85,B 0,C 180,E1 -4619.577,E2 -4619.577} C_VEL
LIN {X 0,Y 523.933,Z 285.225,A -85,B 0,C 180,E1 -4622.45,E2 -4622.45} C_VEL
LIN {X 0,Y 523.919,Z 285.219,A -85,B 0,C 180,E1 -4625.227,E2 -4625.227} C_VEL
LIN {X 0,Y 523.915,Z 285.221,A -85,B 0,C 180,E1 -4628.102,E2 -4628.102} C_VEL
LIN {X 0,Y 523.938,Z 285.218,A -85,B 0,C 180,E1 -4631.092,E2 -4631.092} C_VEL
LIN {X 0,Y 523.929,Z 285.221,A -85,B 0,C 180,E1 -4634.229,E2 -4634.229} C_VEL
LIN {X 0,Y 523.916,Z 285.226,A -85,B 0,C 180,E1 -4636.833,E2 -4636.833} C_VEL
LIN {X 0,Y 523.938,Z 285.223,A -85,B 0,C 180,E1 -4638.908,E2 -4638.908} C_VEL
LIN {X 0,Y 523.914,Z 285.217,A -85,B 0,C 180,E1 -4641.898,E2 -4641.898} C_VEL
LIN {X 0,Y 523.927,Z 285.224,A -85,B 0,C 180,E1 -4644.911,E2 -4644.911} C_VEL
LIN {X 0,Y 523.934,Z 285.215,A -85,B 0,C 180,E1 -4647.68,E2 -4647.68} C_VEL
LIN {X 0,Y 523.953,Z 285.214,A -85,B 0,C 180,E1 -4650.677,E2 -4650.677} C_VEL
LIN {X 0,Y 523.973,Z 285.212,A -85,B 0,C 180,E1 -4653.729,E2 -4653.729} C_VEL
LIN {X 0,Y 523.925,Z 285.214,A -85,B 0,C 180,E1 -4656.27,E2 -4656.27} C_VEL
LIN {X 0,Y 523.944,Z 285.215,A -85,B 0,C 180,E1 -4658.767,E2 -4658.767} C_VEL
LIN {X 0,Y 523.948,Z 285.217,A -85,B 0,C 180,E1 -4661.221,E2 -4661.221} C_VEL
LIN {X 0,Y 523.936,Z 285.222,A -85,B 0,C 180,E1 -4663.639,E2 -4663.639} C_VEL
LIN {X 0,Y 523.938,Z 285.219,A -85,B 0,C 180,E1 -4666.028,E2 -4666.028} C_VEL
LIN {X 0,Y 524.012,Z 285.205,A -85,B 0,C 180,E1 -4668.394,E2 -4668.394} C_VEL
LIN {X 0,Y 524.002,Z 285.213,A -85,B 0,C 180,E1 -4671.516,E2 -4671.516} C_VEL
LIN {X 0,Y 524.078,Z 285.198,A -85,B 0,C 180,E1 -4674.614,E2 -4674.614} C_VEL
LIN {X 0,Y 524.111,Z 285.198,A -85,B 0,C 180,E1 -4677.695,E2 -4677.695} C_VEL
LIN {X 0,Y 524.121,Z 285.192,A -85,B 0,C 180,E1 -4680.768,E2 -4680.768} C_VEL
LIN {X 0,Y 524.071,Z 285.196,A -85,B 0,C 180,E1 -4683.075,E2 -4683.075} C_VEL
LIN {X 0,Y 524.036,Z 285.211,A -85,B 0,C 180,E1 -4686.159,E2 -4686.159} C_VEL
LIN {X 0,Y 524.003,Z 285.213,A -85,B 0,C 180,E1 -4688.484,E2 -4688.484} C_VEL
LIN {X 0,Y 524.002,Z 285.206,A -85,B 0,C 180,E1 -4691.739,E2 -4691.739} C_VEL
LIN {X 0,Y 523.993,Z 285.209,A -85,B 0,C 180,E1 -4695.053,E2 -4695.053} C_VEL
LIN {X 0,Y 523.963,Z 285.213,A -85,B 0,C 180,E1 -4697.969,E2 -4697.969} C_VEL
LIN {X 0,Y 523.972,Z 285.216,A -85,B 0,C 180,E1 -4700.41,E2 -4700.41} C_VEL
LIN {X 0,Y 523.911,Z 285.225,A -85,B 0,C 180,E1 -4702.894,E2 -4702.894} C_VEL
LIN {X 0,Y 523.953,Z 285.215,A -85,B 0,C 180,E1 -4705.419,E2 -4705.419} C_VEL
LIN {X 0,Y 523.968,Z 285.211,A -85,B 0,C 180,E1 -4707.999,E2 -4707.999} C_VEL
LIN {X 0,Y 523.945,Z 285.222,A -85,B 0,C 180,E1 -4710.855,E2 -4710.855} C_VEL
LIN {X 0,Y 523.959,Z 285.214,A -85,B 0,C 180,E1 -4713.735,E2 -4713.735} C_VEL
LIN {X 0,Y 523.904,Z 285.219,A -85,B 0,C 180,E1 -4716.402,E2 -4716.402} C_VEL
LIN {X 0,Y 523.921,Z 285.225,A -85,B 0,C 180,E1 -4719.085,E2 -4719.085} C_VEL
LIN {X 0,Y 523.952,Z 285.214,A -85,B 0,C 180,E1 -4722.119,E2 -4722.119} C_VEL
LIN {X 0,Y 523.943,Z 285.222,A -85,B 0,C 180,E1 -4725.31,E2 -4725.31} C_VEL
LIN {X 0,Y 523.957,Z 285.214,A -85,B 0,C 180,E1 -4728.69,E2 -4728.69} C_VEL
LIN {X 0,Y 523.918,Z 285.22,A -85,B 0,C 180,E1 -4731.081,E2 -4731.081} C_VEL
LIN {X 0,Y 523.902,Z 285.228,A -85,B 0,C 180,E1 -4733.825,E2 -4733.825} C_VEL
LIN {X 0,Y 523.943,Z 285.216,A -85,B 0,C 180,E1 -4736.636,E2 -4736.636} C_VEL
LIN {X 0,Y 523.958,Z 285.217,A -85,B 0,C 180,E1 -4739.356,E2 -4739.356} C_VEL
LIN {X 0,Y 523.978,Z 285.216,A -85,B 0,C 180,E1 -4742.282,E2 -4742.282} C_VEL
LIN {X 0,Y 523.955,Z 285.219,A -85,B 0,C 180,E1 -4744.581,E2 -4744.581} C_VEL
LIN {X 0,Y 523.993,Z 285.3,A -85,B 0,C 180,E1 -4745.481,E2 -4745.481} C_VEL
LIN {X 0,Y 525.362,Z 292.968,A -85,B 0,C 180,E1 -4746.757,E2 -4746.757} C_VEL
LIN {X 0,Y 525,Z 311.46,A -85,B 0,C 180,E1 -4749.632,E2 -4749.632} C_VEL
LIN {X 0,Y 524.54,Z 331.217,A -85,B 0,C 180,E1 -4752.655,E2 -4752.655} C_VEL
LIN {X 0,Y 524.321,Z 345.878,A -85,B 0,C 180,E1 -4754.846,E2 -4754.846} C_VEL
LIN {X 0,Y 525.907,Z 356.631,A -85,B 0,C 180,E1 -4755.041,E2 -4755.041} C_VEL
LIN {X 0,Y 525.491,Z 453.914,A -85,B 0,C 180,E1 -4756.39,E2 -4756.39} C_VEL
LIN {X 0,Y 525.296,Z 467.238,A -85,B 0,C 180,E1 -4756.73,E2 -4756.73} C_VEL
LIN {X 0,Y 525.021,Z 479.435,A -85,B 0,C 180,E1 -4757.19,E2 -4757.19} C_VEL
LIN {X 0,Y 524.807,Z 491.488,A -85,B 0,C 180,E1 -4757.808,E2 -4757.808} C_VEL
LIN {X 0,Y 524.534,Z 503.371,A -85,B 0,C 180,E1 -4758.601,E2 -4758.601} C_VEL
LIN {X 0,Y 524.217,Z 513.837,A -85,B 0,C 180,E1 -4759.475,E2 -4759.475} C_VEL
LIN {X 0,Y 523.985,Z 522.397,A -85,B 0,C 180,E1 -4760.348,E2 -4760.348} C_VEL
LIN {X 0,Y 523.774,Z 530.296,A -85,B 0,C 180,E1 -4761.318,E2 -4761.318} C_VEL
LIN {X 0,Y 523.606,Z 538.012,A -85,B 0,C 180,E1 -4762.48,E2 -4762.48} C_VEL
LIN {X 0,Y 523.484,Z 545.125,A -85,B 0,C 180,E1 -4763.834,E2 -4763.834} C_VEL
LIN {X 0,Y 523.384,Z 549.857,A -85,B 0,C 180,E1 -4764.993,E2 -4764.993} C_VEL
